// TwinCAT 3 PLC project Second_Floor_Totes_ARUP
// ProgramVersion: 3.1.4023.0
// libraries:
//   VisuElemMeter, * (System)
//   VisuElems, * (System)
//   VisuElemsSpecialControls, * (System)
//   VisuElemsWinControls, * (System)
//   VisuElemTextEditor, * (System)
//   VisuInputs, * (System)
//   VisuNativeControl, * (System)
//   Tc2_Standard, * (Beckhoff Automation GmbH)
//   Tc2_System, * (Beckhoff Automation GmbH)
//   Tc2_TcpIp, * (Beckhoff Automation GmbH)
//   Tc2_Utilities, * (Beckhoff Automation GmbH)
//   Tc3_Module, * (Beckhoff Automation GmbH)
// project tree:
//   DUTs/EAP/ E_EAP_PubType.TcDUT, ST_EAP_DEVICE.TcDUT (not stored), ST_EAP_Publisher.TcDUT, ST_EAP_Pub_Variable.TcDUT, ST_EAP_Subscriber.TcDUT (not stored), ST_EAP_Sub_Variable.TcDUT
//   DUTs/ E_EquipType.TcTLEO (not stored), E_StatusCode.TcDUT (not stored), ST_EquipmentStatus.TcDUT (not stored), ST_SafetyState.TcDUT (not stored)
//   DUTs/Messages/ E_EquipmentUpdate.TcTLEO (not stored), E_MessageIds.TcTLEO (not stored), E_TransportComplete.TcDUT (not stored), E_TransportResponse.TcTLEO (not stored), ST_Msg_ConveyorStat.TcDUT (not stored), ST_Msg_EquipStat.TcDUT (not stored)
//   / GlobalTextList.TcGTLO, PlcTask.TcTTO, Visualization Manager.TcVMO (not stored)
//   GVLs/ GVL_EquipArrays.TcGVL, GVL_IO.TcGVL, GVL_Logging.TcGVL, GVL_SorterItems.TcGVL, Onsite_Checklist.TcGVL
//   POUs/ BarCodeReaders.TcPOU, CommStatus.TcPOU, Conveyors.TcPOU, Log_Diverts.TcPOU, MAIN.TcPOU, MsgControl.TcPOU, Photoeyes.TcPOU, ProcessBuffers_6040.TcPOU, ProxSensors.TcPOU, P_PulseCountDist.TcPOU, ServerControl.TcPOU (not stored), Singulation_Control.TcPOU, Solenoids.TcPOU, Sorter.TcPOU, Sorter_P6040.TcPOU, System.TcPOU, SystemSafety.TcPOU
//   POUs/FunctionBlocks/BarCode/ CognexDataMan260.TcPOU (not stored)
//   POUs/FunctionBlocks/Binder/ BinderX_ReleaseControl.TcPOU (not stored), FB_BinderPusher.TcPOU (not stored), FB_Binder_SingulateHold.TcPOU (not stored)
//   POUs/FunctionBlocks/Binder/DUTs/ ST_Binder.TcDUT (not stored), ST_BinderState.TcDUT (not stored), ST_FromBinder.TcDUT (not stored), ST_ToBinder.TcDUT (not stored)
//   POUs/FunctionBlocks/Conveyance/DUTs/ E_ConvType.TcDUT (not stored)
//   POUs/FunctionBlocks/Conveyance/ FB_CnvyrCnfig_1.TcPOU, FB_SleepCntrl.TcPOU (not stored)
//   POUs/FunctionBlocks/Divert/DUTs/ ST_Divert.TcDUT, ST_DivertCfg.TcDUT
//   POUs/FunctionBlocks/Divert/Functions/ FB_ConfirmCheck.TcPOU (not stored), FB_DivertCommission.TcPOU, FB_DivertControl.TcPOU (not stored), FB_DivertDecision.TcPOU, FB_DivertFullMonitor.TcPOU (not stored), FB_DivertLog.TcPOU (not stored)
//   POUs/FunctionBlocks/Encoder/DUTs/ ST_Encoder.TcDUT (not stored)
//   POUs/FunctionBlocks/Encoder/ FB_ProcessEncoder.TcPOU (not stored)
//   POUs/FunctionBlocks/FB_Merge/ E_MergeState.TcDUT (not stored), FB_Merge2.TcPOU (not stored), MergeExample.TcPOU (not stored), ST_MergeSts.TcDUT (not stored)
//   POUs/FunctionBlocks/FB_Merge/Merge Inlet/ FB_MergeInlet.TcPOU (not stored), ST_MergeInlet.TcDUT (not stored), ST_MergeInletCfg.TcDUT (not stored), ST_MergeInletCtrl.TcDUT (not stored), ST_MergeInletSts.TcDUT (not stored)
//   POUs/FunctionBlocks/FB_MotionMerge/ FB_MotionMerge.TcPOU (not stored), MotionMergeExample.TcPOU (not stored), ST_MotionMergeConfig.TcDUT (not stored), ST_MotionMergeItem.TcDUT (not stored)
//   POUs/FunctionBlocks/Item/DUTs/ ST_Item.TcDUT (not stored), ST_ItemBuffer.TcDUT (not stored), ST_ItemBufferFdbk.TcDUT (not stored), ST_ItemLogBuffer.TcDUT (not stored), ST_ItemTemporary.TcDUT (not stored)
//   POUs/FunctionBlocks/Item/ FB_ItemBuffer.TcPOU (not stored), FB_ItemLogBuffer.TcPOU (not stored)
//   POUs/FunctionBlocks/LEDControl/ FB_LEDModeCtrl.TcPOU (not stored), ST_HMILEDMode.TcDUT (not stored), ST_LEDMode.TcDUT (not stored), ST_RGB.TcDUT (not stored)
//   POUs/FunctionBlocks/Logging/ FB_UpdateLog.TcPOU (not stored), ST_LogMsg.TcDUT (not stored)
//   POUs/FunctionBlocks/Metrics/ FB_Metrics.TcPOU (not stored)
//   POUs/FunctionBlocks/Server/Data types/ E_ConnectionSteps.TcDUT (not stored), E_ServerSteps.TcDUT (not stored)
//   POUs/FunctionBlocks/Server/ FB_Server.TcPOU (not stored), FB_ServerApplication.TcPOU (not stored), FB_ServerConnection.TcPOU (not stored)
//   POUs/FunctionBlocks/Server/Helper POUs/ FB_FrameFifo.TcPOU (not stored), FB_LogFifo.TcPOU (not stored)
//   POUs/FunctionBlocks/Singulation/ FB_Singulation.TcPOU (not stored)
//   POUs/FunctionBlocks/Solenoids/Functions/ FB_Solenoid_DA.TcPOU, FB_Solenoid_SA.TcPOU
//   POUs/FunctionBlocks/Sorter/DUTs/ ST_RoundRobin.TcDUT, ST_RoundRobinCfg.TcDUT (not stored), ST_RoundRobinDest.TcDUT (not stored), ST_Sorter.TcDUT, ST_SorterConfig.TcDUT
//   POUs/FunctionBlocks/Sorter/Functions/ FB_FindDestination.TcPOU, FB_SorterLog.TcPOU
//   POUs/FunctionBlocks/Sorter/ ProcessBuffers.TcPOU, SorterExample.TcPOU, SorterProgram.TcPOU (not stored)
//   POUs/FunctionBlocks/Sorter/VISUs/ ArrayInspection.TcVIS (not stored), DiverterTest.TcVIS (not stored), SorterArray.TcVIS
//   POUs/FunctionBlocks/StateControl/ E_OperStateCntrl.TcTLEO (not stored), E_StateCntrl.TcTLEO (not stored), E_StopCodes.TcTLEO (not stored), FB_ManageCodes.TcPOU (not stored), FB_StateCntrl.TcPOU (not stored), ST_StateCntrlPB.TcDUT (not stored), ST_StateCntrlSts.TcDUT (not stored)
//   POUs/FunctionBlocks/Utils/Events/ FB_EventMngr.TcPOU (not stored), FB_Intlks_Latch.TcPOU (not stored), FB_Intlks_NoLatch.TcPOU (not stored), ST_CfgEvents.TcDUT (not stored), ST_EventSts.TcDUT (not stored)
//   POUs/FunctionBlocks/Utils/ FB_AlrtStrtDelay.TcPOU (not stored), FB_EquipCntrl.TcPOU (not stored), FB_Flasher.TcPOU (not stored), FB_FlipFlop.TcPOU (not stored), FB_JamDetect.TcPOU (not stored), FB_PhotoEye.TcPOU (not stored), FB_SystemCntrl.TcPOU, F_CalculateDifference.TcPOU (not stored), F_CalculateIndex.TcPOU (not stored), F_DecIndex.TcPOU (not stored), F_IncIndex.TcPOU (not stored), F_PaddNumber.TcPOU (not stored), IncIndex.TcPOU (not stored), SystemCntrl_Example.TcPOU (not stored)
//   POUs/FunctionBlocks/Utils/Filters/ FB_DigDebnce.TcPOU, FB_DigDebnce_Off.TcPOU (not stored), FB_DigDebnce_On.TcPOU (not stored), F_Clip.TcPOU (not stored)
//   POUs/FunctionBlocks/VFD/DUTs/ DRIVE_STATE.TcTLEO (not stored)
//   POUs/FunctionBlocks/VFD/Functions/ DriveState.TcPOU (not stored), VFD.TcPOU
// real-time tasks:
//   TASK PlcTask: cycle T#10ms, priority 20, ADS port 350
//   TASK BCR_Sync: cycle T#1ms, priority 1, ADS port 301
// I/O:
//   DEVICE Device 1 (RT-Ethernet Protocol), AmsNetId 5.84.5.2.2.1
//   DEVICE Device 2 (TC3 EIP Scanner), AmsNetId 5.84.5.2.3.1
//     BCR_S6040_01 // <INFO> </INFO> <EDS> C:\TwinCAT\3.1\Config\Io\EtherNetIP\0678077313070100.eds </EDS>
//     BCR_S7004_01 // <INFO> </INFO> <EDS> C:\TwinCAT\3.1\Config\Io\EtherNetIP\0678077313070100.eds </EDS>
//   DEVICE Device 3 (EtherCAT), AmsNetId 5.84.5.2.4.1
//     Term 1 (EK1200) [EK1200-5000 EtherCAT Power supply (2A E-Bus)]
//       Term 2 (EL6070-0033) [EL6070-0033 1Ch. Licence key terminal, individual licences]
//       PLC-7021 (EL1008) [EL1008 8Ch. Dig. Input 24V, 3ms]
//       PLC-8051 (EL2008) [EL2008 8Ch. Dig. Output 24V, 0.5A]
//       PLC-8431 (EL1918) [EL1918, 8Ch. Safety Input 24V, TwinSAFE]
//         modules: Module 2 (FSLOGIC)
//       PLC-9071 (EL5152) [EL5152 2Ch. Inc. Encoder]
//       Term 7 (EK1122) [EK1122 2 port EtherCAT junction]
//         RIO-15181 (EP2339-0022) [EP2339-0022 16 Ch. Dig. Input/Output 24V, 0,5A, M12]
//         RIO-16171 (EP2339-0022) [EP2339-0022 16 Ch. Dig. Input/Output 24V, 0,5A, M12]
//         RIO-1181 (EP2339-0022) [EP2339-0022 16 Ch. Dig. Input/Output 24V, 0,5A, M12]
//         RIO-4172 (EP2339-0022) [EP2339-0022 16 Ch. Dig. Input/Output 24V, 0,5A, M12]
//         SRIO-5151 (EP1908) [EP1908, 8 Ch. Safety Input 24V, TwinSAFE ]
//           modules: Module 1 (FSOE)
//         RIO-6171 (EP2339-0022) [EP2339-0022 16 Ch. Dig. Input/Output 24V, 0,5A, M12]
//         RIO-7161 (EP2339-0022) [EP2339-0022 16 Ch. Dig. Input/Output 24V, 0,5A, M12]
//         RIO-8181 (EP2339-0022) [EP2339-0022 16 Ch. Dig. Input/Output 24V, 0,5A, M12]
//       Term 16 (EK1122) [EK1122 2 port EtherCAT junction]
//       Term 17 (EK1122) [EK1122 2 port EtherCAT junction]
//         SRIO-11141 (EP1908) [EP1908, 8 Ch. Safety Input 24V, TwinSAFE ]
//           modules: Module 1 (FSOE)
//         RIO-12171 (EP2339-0022) [EP2339-0022 16 Ch. Dig. Input/Output 24V, 0,5A, M12]
//         Term 18 (EK1100) [EK1100 EtherCAT Coupler (2A E-Bus)]
//           PLC-11021 (EL2008) [EL2008 8Ch. Dig. Output 24V, 0.5A]
//           PLC-11211 (EL2008) [EL2008 8Ch. Dig. Output 24V, 0.5A]
//           PLC-11431 (EL1008) [EL1008 8Ch. Dig. Input 24V, 3ms]
//           PLC-1008 (EL1008) [EL1008 8Ch. Dig. Input 24V, 3ms]
//           PLC-12061 (EL2008) [EL2008 8Ch. Dig. Output 24V, 0.5A]
//           PLC-12461 (EL1008) [EL1008 8Ch. Dig. Input 24V, 3ms]
//           PLC-13051 (EL1918) [EL1918, 8Ch. Safety Input 24V, TwinSAFE]
//             modules: Module 1 (FSOE), Module 2 (FSLOGIC)
//           PLC-13451 (EL2904) [EL2904, 4 Ch. Safety Output 24V, 0.5A, TwinSAFE]
//             modules: Module 1 (FSOES), Module 2 (DO)
//           Term 27 (EK1122) [EK1122 2 port EtherCAT junction]
//             P7040 (Inverter i550 Cabinet) [i550 Cabinet V05.04.xx]
//             P7005 (Inverter i550 Cabinet) [i550 Cabinet V05.04.xx]
//             P6010 (Inverter i550 Cabinet) [i550 Cabinet V05.04.xx]
//             P6045 (Inverter i550 Cabinet) [i550 Cabinet V05.04.xx]
//   DEVICE Communition with 205 (EtherCAT Automation Protocol), AmsNetId 5.84.5.2.5.1
//     Pub_To_205 (Publisher)
//     Sub_To_205 (Subscriber)
// variable links:
//   (this object) <-> Device 3 (EtherCAT)/Term 1 (EK1200)/PLC-8431 (EL1918)
//     Term 1 (EK1200)/Term 17 (EK1122)/SRIO-11141 (EP1908)/Module 1 (FSOE)/FSOE Inputs/FSOE <-> ConnectionOutputs/Message_33 RxPDO
//     Term 1 (EK1200)/Term 7 (EK1122)/SRIO-5151 (EP1908)/Module 1 (FSOE)/FSOE Inputs/FSOE <-> ConnectionOutputs/Message_32 RxPDO
//     Term 1 (EK1200)/Term 17 (EK1122)/SRIO-11141 (EP1908)/Module 1 (FSOE)/FSOE Outputs/FSOE <-> ConnectionInputs/Message_33 TxPDO
//     Term 1 (EK1200)/Term 7 (EK1122)/SRIO-5151 (EP1908)/Module 1 (FSOE)/FSOE Outputs/FSOE <-> ConnectionInputs/Message_32 TxPDO
//     Term 1 (EK1200)/Term 17 (EK1122)/Term 18 (EK1100)/PLC-13051 (EL1918)/Module 1 (FSOE)/FSoE Inputs/FSOE <-> ConnectionOutputs/Message_30 RxPDO
//     Term 1 (EK1200)/Term 17 (EK1122)/Term 18 (EK1100)/PLC-13051 (EL1918)/Module 1 (FSOE)/FSoE Outputs/FSOE <-> ConnectionInputs/Message_30 TxPDO
//     Term 1 (EK1200)/Term 17 (EK1122)/Term 18 (EK1100)/PLC-13451 (EL2904)/Module 1 (FSOES)/RxPDO/FSOE <-> ConnectionInputs/Message_31 TxPDO
//     Term 1 (EK1200)/Term 17 (EK1122)/Term 18 (EK1100)/PLC-13451 (EL2904)/Module 1 (FSOES)/TxPDO/FSOE <-> ConnectionOutputs/Message_31 RxPDO
//   (this object) <-> Device 3 (EtherCAT)/Term 1 (EK1200)/Term 17 (EK1122)/SRIO-11141 (EP1908)
//     Term 1 (EK1200)/PLC-8431 (EL1918)/ConnectionInputs/Message_33 TxPDO <-> Module 1 (FSOE)/FSOE Outputs/FSOE
//     Term 1 (EK1200)/PLC-8431 (EL1918)/ConnectionOutputs/Message_33 RxPDO <-> Module 1 (FSOE)/FSOE Inputs/FSOE
//   (this object) <-> Device 3 (EtherCAT)/Term 1 (EK1200)/Term 17 (EK1122)/Term 18 (EK1100)/PLC-13051 (EL1918)
//     Term 1 (EK1200)/PLC-8431 (EL1918)/ConnectionInputs/Message_30 TxPDO <-> Module 1 (FSOE)/FSoE Outputs/FSOE
//     Term 1 (EK1200)/PLC-8431 (EL1918)/ConnectionOutputs/Message_30 RxPDO <-> Module 1 (FSOE)/FSoE Inputs/FSOE
//   (this object) <-> Device 3 (EtherCAT)/Term 1 (EK1200)/Term 17 (EK1122)/Term 18 (EK1100)/PLC-13451 (EL2904)
//     Term 1 (EK1200)/PLC-8431 (EL1918)/ConnectionInputs/Message_31 TxPDO <-> Module 1 (FSOES)/RxPDO/FSOE
//     Term 1 (EK1200)/PLC-8431 (EL1918)/ConnectionOutputs/Message_31 RxPDO <-> Module 1 (FSOES)/TxPDO/FSOE
//   (this object) <-> Device 3 (EtherCAT)/Term 1 (EK1200)/Term 7 (EK1122)/SRIO-5151 (EP1908)
//     Term 1 (EK1200)/PLC-8431 (EL1918)/ConnectionInputs/Message_32 TxPDO <-> Module 1 (FSOE)/FSOE Outputs/FSOE
//     Term 1 (EK1200)/PLC-8431 (EL1918)/ConnectionOutputs/Message_32 RxPDO <-> Module 1 (FSOE)/FSOE Inputs/FSOE
//   Second_Floor_Totes_ARUP Instance <-> Communition with 205 (EtherCAT Automation Protocol)
//     PlcTask Inputs/MAIN.EAP_205.DevState <-> Inputs/DevState
//     PlcTask Outputs/MAIN.EAP_205.DevCtrl <-> Outputs/DevCtrl
//   Second_Floor_Totes_ARUP Instance <-> Communition with 205 (EtherCAT Automation Protocol)/Pub_To_205 (Publisher)
//     PlcTask Inputs/MAIN.EAP_205.Publisher.FrameState <-> Inputs/FrameState
//     PlcTask Inputs/MAIN.EAP_205.Publisher.Variables[0].VarState <-> To205_P6005_IsRunning/Inputs/VarState
//     PlcTask Inputs/MAIN.EAP_205.Publisher.Variables[1].VarState <-> To205_P7045_SendingProduct/Inputs/VarState
//     PlcTask Outputs/GVL_IO.To205_P6005_IsRunning <-> To205_P6005_IsRunning/Outputs/VarData
//     PlcTask Outputs/GVL_IO.To205_P7045_SendingProduct <-> To205_P7045_SendingProduct/Outputs/VarData
//     PlcTask Outputs/MAIN.EAP_205.Publisher.FrameCtrl <-> Outputs/FrameCtrl
//     PlcTask Outputs/MAIN.EAP_205.Publisher.IPAddr <-> Outputs/IpAddr
//     PlcTask Outputs/MAIN.EAP_205.Publisher.Variables[0].VarCtrl <-> To205_P6005_IsRunning/Outputs/VarCtrl
//     PlcTask Outputs/MAIN.EAP_205.Publisher.Variables[0].VarID <-> To205_P6005_IsRunning/Outputs/VarId
//     PlcTask Outputs/MAIN.EAP_205.Publisher.Variables[1].VarCtrl <-> To205_P7045_SendingProduct/Outputs/VarCtrl
//     PlcTask Outputs/MAIN.EAP_205.Publisher.Variables[1].VarID <-> To205_P7045_SendingProduct/Outputs/VarId
//   Second_Floor_Totes_ARUP Instance <-> Communition with 205 (EtherCAT Automation Protocol)/Sub_To_205 (Subscriber)
//     PlcTask Inputs/GVL_IO.From205_P2012_IsRunning <-> From205_P2012_IsRunning/Inputs/VarData
//     PlcTask Inputs/GVL_IO.From205_P3130_SendingProduct <-> From205_P3130_SendingProduct/Inputs/VarData
//     PlcTask Inputs/MAIN.EAP_205.Subscriber.FrameState <-> Inputs/FrameState
//     PlcTask Inputs/MAIN.EAP_205.Subscriber.Variables[0].CycleIndex <-> From205_P2012_IsRunning/Inputs/CycleIndex
//     PlcTask Inputs/MAIN.EAP_205.Subscriber.Variables[0].Quality <-> From205_P2012_IsRunning/Inputs/Quality
//     PlcTask Inputs/MAIN.EAP_205.Subscriber.Variables[0].VarState <-> From205_P2012_IsRunning/Inputs/VarState
//     PlcTask Inputs/MAIN.EAP_205.Subscriber.Variables[1].CycleIndex <-> From205_P3130_SendingProduct/Inputs/CycleIndex
//     PlcTask Inputs/MAIN.EAP_205.Subscriber.Variables[1].Quality <-> From205_P3130_SendingProduct/Inputs/Quality
//     PlcTask Inputs/MAIN.EAP_205.Subscriber.Variables[1].VarState <-> From205_P3130_SendingProduct/Inputs/VarState
//     PlcTask Outputs/MAIN.EAP_205.Subscriber.FrameCtrl <-> Outputs/FrameCtrl
//     PlcTask Outputs/MAIN.EAP_205.Subscriber.Variables[0].VarCtrl <-> From205_P2012_IsRunning/Outputs/VarCtrl
//     PlcTask Outputs/MAIN.EAP_205.Subscriber.Variables[0].VarId <-> From205_P2012_IsRunning/Outputs/VarId
//     PlcTask Outputs/MAIN.EAP_205.Subscriber.Variables[1].VarCtrl <-> From205_P3130_SendingProduct/Outputs/VarCtrl
//     PlcTask Outputs/MAIN.EAP_205.Subscriber.Variables[1].VarId <-> From205_P3130_SendingProduct/Outputs/VarId
//   Second_Floor_Totes_ARUP Instance <-> Device 1 (RT-Ethernet Protocol)
//     PlcTask Inputs/GVL_IO.EthernetAdapter_State <-> Inputs/DevState
//   Second_Floor_Totes_ARUP Instance <-> Device 2 (TC3 EIP Scanner)/BCR_S6040_01
//     PlcTask Inputs/BarCodeReaders.BCR_S6040_01.Acquiring <-> Connection 1 (Input/Output)/Inputs/Acquiring
//     PlcTask Inputs/BarCodeReaders.BCR_S6040_01.DecodeComplete <-> Connection 1 (Input/Output)/Inputs/Decode Complete
//     PlcTask Inputs/BarCodeReaders.BCR_S6040_01.Decoding <-> Connection 1 (Input/Output)/Inputs/Decoding
//     PlcTask Inputs/BarCodeReaders.BCR_S6040_01.DeviceState <-> Inputs/State
//     PlcTask Inputs/BarCodeReaders.BCR_S6040_01.ResultCode <-> Connection 1 (Input/Output)/Inputs/Result Code
//     PlcTask Inputs/BarCodeReaders.BCR_S6040_01.ResultData[0] <-> Connection 1 (Input/Output)/Inputs/Result Data
//     PlcTask Inputs/BarCodeReaders.BCR_S6040_01.ResultData[10] <-> Connection 1 (Input/Output)/Inputs/Result Data_10
//     PlcTask Inputs/BarCodeReaders.BCR_S6040_01.ResultData[11] <-> Connection 1 (Input/Output)/Inputs/Result Data_11
//     PlcTask Inputs/BarCodeReaders.BCR_S6040_01.ResultData[12] <-> Connection 1 (Input/Output)/Inputs/Result Data_12
//     PlcTask Inputs/BarCodeReaders.BCR_S6040_01.ResultData[13] <-> Connection 1 (Input/Output)/Inputs/Result Data_13
//     PlcTask Inputs/BarCodeReaders.BCR_S6040_01.ResultData[14] <-> Connection 1 (Input/Output)/Inputs/Result Data_14
//     PlcTask Inputs/BarCodeReaders.BCR_S6040_01.ResultData[15] <-> Connection 1 (Input/Output)/Inputs/Result Data_15
//     PlcTask Inputs/BarCodeReaders.BCR_S6040_01.ResultData[16] <-> Connection 1 (Input/Output)/Inputs/Result Data_16
//     PlcTask Inputs/BarCodeReaders.BCR_S6040_01.ResultData[1] <-> Connection 1 (Input/Output)/Inputs/Result Data_1
//     PlcTask Inputs/BarCodeReaders.BCR_S6040_01.ResultData[2] <-> Connection 1 (Input/Output)/Inputs/Result Data_2
//     PlcTask Inputs/BarCodeReaders.BCR_S6040_01.ResultData[3] <-> Connection 1 (Input/Output)/Inputs/Result Data_3
//     PlcTask Inputs/BarCodeReaders.BCR_S6040_01.ResultData[4] <-> Connection 1 (Input/Output)/Inputs/Result Data_4
//     PlcTask Inputs/BarCodeReaders.BCR_S6040_01.ResultData[5] <-> Connection 1 (Input/Output)/Inputs/Result Data_5
//     PlcTask Inputs/BarCodeReaders.BCR_S6040_01.ResultData[6] <-> Connection 1 (Input/Output)/Inputs/Result Data_6
//     PlcTask Inputs/BarCodeReaders.BCR_S6040_01.ResultData[7] <-> Connection 1 (Input/Output)/Inputs/Result Data_7
//     PlcTask Inputs/BarCodeReaders.BCR_S6040_01.ResultData[8] <-> Connection 1 (Input/Output)/Inputs/Result Data_8
//     PlcTask Inputs/BarCodeReaders.BCR_S6040_01.ResultData[9] <-> Connection 1 (Input/Output)/Inputs/Result Data_9
//     PlcTask Inputs/BarCodeReaders.BCR_S6040_01.ResultID <-> Connection 1 (Input/Output)/Inputs/Result ID
//     PlcTask Inputs/BarCodeReaders.BCR_S6040_01.ResultLength <-> Connection 1 (Input/Output)/Inputs/Result Length
//     PlcTask Inputs/BarCodeReaders.BCR_S6040_01.ResultsAvail <-> Connection 1 (Input/Output)/Inputs/Results Available
//     PlcTask Inputs/BarCodeReaders.BCR_S6040_01.TriggerAck <-> Connection 1 (Input/Output)/Inputs/Trigger Ack
//     PlcTask Inputs/BarCodeReaders.BCR_S6040_01.TriggerID <-> Connection 1 (Input/Output)/Inputs/Trigger ID
//     PlcTask Inputs/BarCodeReaders.BCR_S6040_01.TriggerReady <-> Connection 1 (Input/Output)/Inputs/Trigger Ready
//     PlcTask Outputs/BarCodeReaders.BCR_S6040_01.ResultsAck <-> Connection 1 (Input/Output)/Outputs/Results Ack
//     PlcTask Outputs/BarCodeReaders.BCR_S6040_01.Trigger <-> Connection 1 (Input/Output)/Outputs/Trigger
//     PlcTask Outputs/BarCodeReaders.BCR_S6040_01.TriggerEnable <-> Connection 1 (Input/Output)/Outputs/Trigger Enable
//   Second_Floor_Totes_ARUP Instance <-> Device 2 (TC3 EIP Scanner)/BCR_S7004_01
//     PlcTask Inputs/BarCodeReaders.BCR_S7004_01.Acquiring <-> Connection 2 (Input/Output)/Inputs/Acquiring
//     PlcTask Inputs/BarCodeReaders.BCR_S7004_01.DecodeComplete <-> Connection 2 (Input/Output)/Inputs/Decode Complete
//     PlcTask Inputs/BarCodeReaders.BCR_S7004_01.Decoding <-> Connection 2 (Input/Output)/Inputs/Decoding
//     PlcTask Inputs/BarCodeReaders.BCR_S7004_01.DeviceState <-> Inputs/State
//     PlcTask Inputs/BarCodeReaders.BCR_S7004_01.ResultCode <-> Connection 2 (Input/Output)/Inputs/Result Code
//     PlcTask Inputs/BarCodeReaders.BCR_S7004_01.ResultData[0] <-> Connection 2 (Input/Output)/Inputs/Result Data
//     PlcTask Inputs/BarCodeReaders.BCR_S7004_01.ResultData[10] <-> Connection 2 (Input/Output)/Inputs/Result Data_10
//     PlcTask Inputs/BarCodeReaders.BCR_S7004_01.ResultData[11] <-> Connection 2 (Input/Output)/Inputs/Result Data_11
//     PlcTask Inputs/BarCodeReaders.BCR_S7004_01.ResultData[12] <-> Connection 2 (Input/Output)/Inputs/Result Data_12
//     PlcTask Inputs/BarCodeReaders.BCR_S7004_01.ResultData[13] <-> Connection 2 (Input/Output)/Inputs/Result Data_13
//     PlcTask Inputs/BarCodeReaders.BCR_S7004_01.ResultData[14] <-> Connection 2 (Input/Output)/Inputs/Result Data_14
//     PlcTask Inputs/BarCodeReaders.BCR_S7004_01.ResultData[15] <-> Connection 2 (Input/Output)/Inputs/Result Data_15
//     PlcTask Inputs/BarCodeReaders.BCR_S7004_01.ResultData[16] <-> Connection 2 (Input/Output)/Inputs/Result Data_16
//     PlcTask Inputs/BarCodeReaders.BCR_S7004_01.ResultData[1] <-> Connection 2 (Input/Output)/Inputs/Result Data_1
//     PlcTask Inputs/BarCodeReaders.BCR_S7004_01.ResultData[2] <-> Connection 2 (Input/Output)/Inputs/Result Data_2
//     PlcTask Inputs/BarCodeReaders.BCR_S7004_01.ResultData[3] <-> Connection 2 (Input/Output)/Inputs/Result Data_3
//     PlcTask Inputs/BarCodeReaders.BCR_S7004_01.ResultData[4] <-> Connection 2 (Input/Output)/Inputs/Result Data_4
//     PlcTask Inputs/BarCodeReaders.BCR_S7004_01.ResultData[5] <-> Connection 2 (Input/Output)/Inputs/Result Data_5
//     PlcTask Inputs/BarCodeReaders.BCR_S7004_01.ResultData[6] <-> Connection 2 (Input/Output)/Inputs/Result Data_6
//     PlcTask Inputs/BarCodeReaders.BCR_S7004_01.ResultData[7] <-> Connection 2 (Input/Output)/Inputs/Result Data_7
//     PlcTask Inputs/BarCodeReaders.BCR_S7004_01.ResultData[8] <-> Connection 2 (Input/Output)/Inputs/Result Data_8
//     PlcTask Inputs/BarCodeReaders.BCR_S7004_01.ResultData[9] <-> Connection 2 (Input/Output)/Inputs/Result Data_9
//     PlcTask Inputs/BarCodeReaders.BCR_S7004_01.ResultID <-> Connection 2 (Input/Output)/Inputs/Result ID
//     PlcTask Inputs/BarCodeReaders.BCR_S7004_01.ResultLength <-> Connection 2 (Input/Output)/Inputs/Result Length
//     PlcTask Inputs/BarCodeReaders.BCR_S7004_01.ResultsAvail <-> Connection 2 (Input/Output)/Inputs/Results Available
//     PlcTask Inputs/BarCodeReaders.BCR_S7004_01.TriggerAck <-> Connection 2 (Input/Output)/Inputs/Trigger Ack
//     PlcTask Inputs/BarCodeReaders.BCR_S7004_01.TriggerID <-> Connection 2 (Input/Output)/Inputs/Trigger ID
//     PlcTask Inputs/BarCodeReaders.BCR_S7004_01.TriggerReady <-> Connection 2 (Input/Output)/Inputs/Trigger Ready
//     PlcTask Outputs/BarCodeReaders.BCR_S7004_01.ResultsAck <-> Connection 2 (Input/Output)/Outputs/Results Ack
//     PlcTask Outputs/BarCodeReaders.BCR_S7004_01.Trigger <-> Connection 2 (Input/Output)/Outputs/Trigger
//     PlcTask Outputs/BarCodeReaders.BCR_S7004_01.TriggerEnable <-> Connection 2 (Input/Output)/Outputs/Trigger Enable
//   Second_Floor_Totes_ARUP Instance <-> Device 3 (EtherCAT)/Term 1 (EK1200)/PLC-7021 (EL1008)
//     PlcTask Inputs/GVL_IO.PB_SysReset <-> Channel 3/Reset PB
//     PlcTask Inputs/GVL_IO.PB_SysStart <-> Channel 1/Start PB
//     PlcTask Inputs/GVL_IO.PB_SysStop <-> Channel 2/Stop PB
//   Second_Floor_Totes_ARUP Instance <-> Device 3 (EtherCAT)/Term 1 (EK1200)/PLC-8051 (EL2008)
//     PlcTask Outputs/GVL_IO.HornMainPanel <-> Channel 1/Horn
//     PlcTask Outputs/GVL_IO.LT_MainPanelStack_Green <-> Channel 4/LT-8111
//     PlcTask Outputs/GVL_IO.LT_MainPanelStack_Red <-> Channel 2/LT-8071
//     PlcTask Outputs/GVL_IO.LT_MainPanelStack_Yellow <-> Channel 3/LT-8091
//   Second_Floor_Totes_ARUP Instance <-> Device 3 (EtherCAT)/Term 1 (EK1200)/PLC-8431 (EL1918)
//     PlcTask Inputs/GVL_IO.PanelEstop_OK <-> StandardInputs/Standard Out Var 9
//     PlcTask Inputs/GVL_IO.Remote_PullCord6040_OK <-> StandardInputs/Standard Out Var 10
//     PlcTask Inputs/GVL_IO.Remote_PullCord7004_OK <-> StandardInputs/Standard Out Var 11
//     PlcTask Inputs/SystemSafety.Safety_SystemEstopsOK <-> StandardInputs/Standard Out Var 15
//     PlcTask Inputs/SystemSafety.SecondFloorShaft_Estop_OK <-> StandardInputs/Standard Out Var 36
//     PlcTask Inputs/SystemSafety.System_SafetyState.ComErr <-> StandardInputs/Standard Out Var 16
//     PlcTask Inputs/SystemSafety.System_SafetyState.FBErr <-> StandardInputs/Standard Out Var 17
//     PlcTask Inputs/SystemSafety.System_SafetyState.InRun <-> StandardInputs/Standard Out Var 38
//     PlcTask Inputs/SystemSafety.System_SafetyState.OtherErr <-> StandardInputs/Standard Out Var 18
//     PlcTask Inputs/SystemSafety.ThirdFloorShaft_Estop_OK <-> StandardInputs/Standard Out Var 37
//     PlcTask Outputs/SystemSafety.System_SafetyState.CommErrAck <-> StandardOutputs/Standard In Var 35
//     PlcTask Outputs/SystemSafety.System_SafetyState.ErrAck <-> StandardOutputs/Standard In Var 1
//     PlcTask Outputs/SystemSafety.System_SafetyState.Reset <-> StandardOutputs/Standard In Var 5
//     PlcTask Outputs/SystemSafety.System_SafetyState.Run <-> StandardOutputs/Standard In Var 2
//   Second_Floor_Totes_ARUP Instance <-> Device 3 (EtherCAT)/Term 1 (EK1200)/PLC-9071 (EL5152)
//     PlcTask Inputs/GVL_IO.ENC_9021_Period <-> ENC Period Channel 1/Period value
//     PlcTask Inputs/GVL_IO.ENC_9021_Raw <-> ENC Status compact Channel 1/Counter value
//   Second_Floor_Totes_ARUP Instance <-> Device 3 (EtherCAT)/Term 1 (EK1200)/Term 17 (EK1122)/RIO-12171 (EP2339-0022)
//     PlcTask Inputs/GVL_IO.DS_P7004 <-> Channel 9/P7004 Motor Disconnect
//     PlcTask Inputs/GVL_IO.DS_P7005 <-> Channel 8/P7005 Motor Discconnect
//     PlcTask Inputs/GVL_IO.DS_P7010 <-> Channel 11/P7010 Motor Discconnect
//     PlcTask Inputs/GVL_IO.PB_RemoteReset_12181 <-> Channel 4/PB-12181
//     PlcTask Inputs/GVL_IO.RIO12171_WcState <-> WcState/WcState
//     PlcTask Inputs/PhotoEyes.PE_12221.In_PE <-> Channel 5/PE-12221
//     PlcTask Inputs/PhotoEyes.PE_12261.In_PE <-> Channel 6/PE-12261
//     PlcTask Inputs/PhotoEyes.PE_12301.In_PE <-> Channel 7/PE-12301
//     PlcTask Inputs/PhotoEyes.PE_12231.In_PE <-> Channel 12/PE12231
//     PlcTask Outputs/GVL_IO.LT_12121_Red <-> Channel 17/LT-12121
//     PlcTask Outputs/GVL_IO.LT_12131_Yellow <-> Channel 18/LT-12131
//     PlcTask Outputs/GVL_IO.LT_12161_Green <-> Channel 19/LT-12161
//   Second_Floor_Totes_ARUP Instance <-> Device 3 (EtherCAT)/Term 1 (EK1200)/Term 17 (EK1122)/SRIO-11141 (EP1908)
//     PlcTask Inputs/GVL_IO.RIO11141_WcState <-> WcState/WcState
//   Second_Floor_Totes_ARUP Instance <-> Device 3 (EtherCAT)/Term 1 (EK1200)/Term 17 (EK1122)/Term 18 (EK1100)/PLC-1008 (EL1008)
//     PlcTask Inputs/GVL_IO.P6005_Faulted <-> Channel 1/P6005 Faulted
//     PlcTask Inputs/GVL_IO.P6015_Faulted <-> Channel 2/P6015 Faulted
//     PlcTask Inputs/GVL_IO.P6020_Faulted <-> Channel 3/P6020 Faulted
//     PlcTask Inputs/GVL_IO.P6025_Faulted <-> Channel 4/P6025 Faulted
//     PlcTask Inputs/GVL_IO.P6030_Faulted <-> Channel 5/P6030 Faulted
//     PlcTask Inputs/GVL_IO.P6035_Faulted <-> Channel 6/P6035 Faulted
//     PlcTask Inputs/GVL_IO.P6040_Faulted <-> Channel 7/P6040 Faulted
//   Second_Floor_Totes_ARUP Instance <-> Device 3 (EtherCAT)/Term 1 (EK1200)/Term 17 (EK1122)/Term 18 (EK1100)/PLC-11021 (EL2008)
//     PlcTask Outputs/GVL_IO.P7004_RUN <-> Channel 1/P7004 RUN
//     PlcTask Outputs/GVL_IO.P7010_RUN <-> Channel 2/P7010 RUN
//     PlcTask Outputs/GVL_IO.P7015_RUN <-> Channel 3/P7015 RUN
//     PlcTask Outputs/GVL_IO.P7020_RUN <-> Channel 4/P7020 RUN
//     PlcTask Outputs/GVL_IO.P7025_RUN <-> Channel 5/P7025 RUN
//     PlcTask Outputs/GVL_IO.P7030_RUN <-> Channel 6/P7030 RUN
//     PlcTask Outputs/GVL_IO.P7035_RUN <-> Channel 7/P7035 RUN
//     PlcTask Outputs/GVL_IO.P7045_RUN <-> Channel 8/P7045 RUN
//   Second_Floor_Totes_ARUP Instance <-> Device 3 (EtherCAT)/Term 1 (EK1200)/Term 17 (EK1122)/Term 18 (EK1100)/PLC-11211 (EL2008)
//     PlcTask Outputs/GVL_IO.P6005_RUN <-> Channel 1/P6005 RUN
//     PlcTask Outputs/GVL_IO.P6015_RUN <-> Channel 2/P6015 RUN
//     PlcTask Outputs/GVL_IO.P6020_RUN <-> Channel 3/P6020 RUN
//     PlcTask Outputs/GVL_IO.P6025_RUN <-> Channel 4/P6025 RUN
//     PlcTask Outputs/GVL_IO.P6030_RUN <-> Channel 5/P6030 RUN
//     PlcTask Outputs/GVL_IO.P6035_RUN <-> Channel 6/P6035 RUN
//     PlcTask Outputs/GVL_IO.P6040_RUN <-> Channel 7/P6040 RUN
//   Second_Floor_Totes_ARUP Instance <-> Device 3 (EtherCAT)/Term 1 (EK1200)/Term 17 (EK1122)/Term 18 (EK1100)/PLC-11431 (EL1008)
//     PlcTask Inputs/GVL_IO.P7004_Faulted <-> Channel 1/P7004 Faulted
//     PlcTask Inputs/GVL_IO.P7010_Faulted <-> Channel 2/P7010 Faulted
//     PlcTask Inputs/GVL_IO.P7015_Faulted <-> Channel 3/P7015 Faulted
//     PlcTask Inputs/GVL_IO.P7020_Faulted <-> Channel 4/P7020 Faulted
//     PlcTask Inputs/GVL_IO.P7025_Faulted <-> Channel 5/P7025 Faulted
//     PlcTask Inputs/GVL_IO.P7030_Faulted <-> Channel 6/P7030 Faulted
//     PlcTask Inputs/GVL_IO.P7035_Faulted <-> Channel 7/P7035 Faulted
//     PlcTask Inputs/GVL_IO.P7045_Faulted <-> Channel 8/P7045 Faulted
//   Second_Floor_Totes_ARUP Instance <-> Device 3 (EtherCAT)/Term 1 (EK1200)/Term 17 (EK1122)/Term 18 (EK1100)/Term 27 (EK1122)/P6010 (Inverter i550 Cabinet)
//     PlcTask Inputs/Conveyors.P6010_VFD.ActualVelocity <-> TPDO (A) Velocity/Actual speed
//     PlcTask Inputs/Conveyors.P6010_VFD.StatusWord <-> TPDO (A) Velocity/CiA status word
//     PlcTask Outputs/Conveyors.P6010_VFD.ControlWord <-> RPDO (A) Velocity/CiA control word
//     PlcTask Outputs/Conveyors.P6010_VFD.TargetVelocity <-> RPDO (A) Velocity/Set speed
//   Second_Floor_Totes_ARUP Instance <-> Device 3 (EtherCAT)/Term 1 (EK1200)/Term 17 (EK1122)/Term 18 (EK1100)/Term 27 (EK1122)/P6045 (Inverter i550 Cabinet)
//     PlcTask Inputs/Conveyors.P6045_VFD.ActualVelocity <-> TPDO (A) Velocity/Actual speed
//     PlcTask Inputs/Conveyors.P6045_VFD.StatusWord <-> TPDO (A) Velocity/CiA status word
//     PlcTask Outputs/Conveyors.P6045_VFD.ControlWord <-> RPDO (A) Velocity/CiA control word
//     PlcTask Outputs/Conveyors.P6045_VFD.TargetVelocity <-> RPDO (A) Velocity/Set speed
//   Second_Floor_Totes_ARUP Instance <-> Device 3 (EtherCAT)/Term 1 (EK1200)/Term 17 (EK1122)/Term 18 (EK1100)/Term 27 (EK1122)/P7005 (Inverter i550 Cabinet)
//     PlcTask Inputs/Conveyors.P7005_VFD.ActualVelocity <-> TPDO (A) Velocity/Actual speed
//     PlcTask Inputs/Conveyors.P7005_VFD.StatusWord <-> TPDO (A) Velocity/CiA status word
//     PlcTask Outputs/Conveyors.P7005_VFD.ControlWord <-> RPDO (A) Velocity/CiA control word
//     PlcTask Outputs/Conveyors.P7005_VFD.TargetVelocity <-> RPDO (A) Velocity/Set speed
//   Second_Floor_Totes_ARUP Instance <-> Device 3 (EtherCAT)/Term 1 (EK1200)/Term 17 (EK1122)/Term 18 (EK1100)/Term 27 (EK1122)/P7040 (Inverter i550 Cabinet)
//     PlcTask Inputs/Conveyors.P7040_VFD.ActualVelocity <-> TPDO (A) Velocity/Actual speed
//     PlcTask Inputs/Conveyors.P7040_VFD.StatusWord <-> TPDO (A) Velocity/CiA status word
//     PlcTask Outputs/Conveyors.P7040_VFD.ControlWord <-> RPDO (A) Velocity/CiA control word
//     PlcTask Outputs/Conveyors.P7040_VFD.TargetVelocity <-> RPDO (A) Velocity/Set speed
//   Second_Floor_Totes_ARUP Instance <-> Device 3 (EtherCAT)/Term 1 (EK1200)/Term 7 (EK1122)/RIO-1181 (EP2339-0022)
//     PlcTask Inputs/GVL_IO.DS_P6005 <-> Channel 14/P6005 Motor Disconnect
//     PlcTask Inputs/GVL_IO.DS_P6015 <-> Channel 10/P6015 Motor Disconnect
//     PlcTask Inputs/GVL_IO.DS_P6010 <-> Channel 12/P6010 Motor Disconnect
//     PlcTask Inputs/GVL_IO.DS_P6020 <-> Channel 4/P6020 Dissconnect
//     PlcTask Inputs/GVL_IO.RIO1181_WcState <-> WcState/WcState
//     PlcTask Inputs/PhotoEyes.PE_1081.In_PE <-> Channel 9/PE-1081
//     PlcTask Inputs/PhotoEyes.PE_1161.In_PE <-> Channel 3/PE-1161
//     PlcTask Inputs/PhotoEyes.PE_1162.In_PE <-> Channel 11/PE-1162
//     PlcTask Inputs/PhotoEyes.PE_1231.In_PE <-> Channel 5/PE-1231
//     PlcTask Inputs/PhotoEyes.PE_1232.In_PE <-> Channel 13/PE-1232
//     PlcTask Inputs/ProxSensors.In_PX_1281_Extended <-> Channel 6/PX-1281
//   Second_Floor_Totes_ARUP Instance <-> Device 3 (EtherCAT)/Term 1 (EK1200)/Term 7 (EK1122)/RIO-15181 (EP2339-0022)
//     PlcTask Inputs/GVL_IO.DS_P7015 <-> Channel 2/P7015 Motor Disconnect
//     PlcTask Inputs/GVL_IO.DS_P7020 <-> Channel 4/P7020 Motor Disconnect
//     PlcTask Inputs/GVL_IO.DS_P7025 <-> Channel 6/P7025 Motor Disconnect
//     PlcTask Inputs/GVL_IO.RIO15181_WcState <-> WcState/WcState
//     PlcTask Inputs/PhotoEyes.PE_15121.In_PE <-> Channel 1/PE-15121
//     PlcTask Inputs/PhotoEyes.PE_15181.In_PE <-> Channel 3/PE-15181
//     PlcTask Inputs/PhotoEyes.PE_15261.In_PE <-> Channel 5/PE-15261
//   Second_Floor_Totes_ARUP Instance <-> Device 3 (EtherCAT)/Term 1 (EK1200)/Term 7 (EK1122)/RIO-16171 (EP2339-0022)
//     PlcTask Inputs/GVL_IO.DS_P7030 <-> Channel 2/P7030 Motor Disconnect
//     PlcTask Inputs/GVL_IO.DS_P7035 <-> Channel 8/P7035 Motor Discconnect
//     PlcTask Inputs/GVL_IO.DS_P7040 <-> Channel 10/P7040 Motor Discconnect
//     PlcTask Inputs/GVL_IO.DS_P7045 <-> Channel 12/P7045 Motor discconnect
//     PlcTask Inputs/GVL_IO.RIO16171_WcState <-> WcState/WcState
//     PlcTask Inputs/PhotoEyes.PE_16111.In_PE <-> Channel 1/PE-16111
//     PlcTask Inputs/PhotoEyes.PE_16131.In_PE <-> Channel 9/PE-16131
//     PlcTask Inputs/PhotoEyes.PE_16181.In_PE <-> Channel 3/PE-16181
//     PlcTask Inputs/PhotoEyes.PE_16201.In_PE <-> Channel 11/PE-16201
//     PlcTask Inputs/PhotoEyes.PE_16301.In_PE <-> Channel 7/PE-16301
//     PlcTask Inputs/ProxSensors.In_PX_16231_Extended <-> Channel 5/PX-16231
//   Second_Floor_Totes_ARUP Instance <-> Device 3 (EtherCAT)/Term 1 (EK1200)/Term 7 (EK1122)/RIO-4172 (EP2339-0022)
//     PlcTask Inputs/GVL_IO.DS_P6025 <-> Channel 10/P6025 Motor disconnect
//     PlcTask Inputs/GVL_IO.DS_P6030 <-> Channel 8/P6030 Motor Discconnect
//     PlcTask Inputs/GVL_IO.DS_P6035 <-> Channel 6/P6035 Motor Disconnect
//     PlcTask Inputs/GVL_IO.DS_P6045 <-> Channel 2/P6045 Motor Discconnect
//     PlcTask Inputs/GVL_IO.RIO4172_WcState <-> WcState/WcState
//     PlcTask Inputs/PhotoEyes.PE_4071.In_PE <-> Channel 1/PE-4071
//     PlcTask Inputs/PhotoEyes.PE_4121.In_PE <-> Channel 9/PE-4121
//     PlcTask Inputs/PhotoEyes.PE_4201.In_PE <-> Channel 5/PE-4201
//     PlcTask Inputs/PhotoEyes.PE_4271.In_PE <-> Channel 7/PE-4271
//   Second_Floor_Totes_ARUP Instance <-> Device 3 (EtherCAT)/Term 1 (EK1200)/Term 7 (EK1122)/RIO-6171 (EP2339-0022)
//     PlcTask Inputs/GVL_IO.RIO6171_WcState <-> WcState/WcState
//     PlcTask Inputs/PhotoEyes.PE_6181.In_PE <-> Channel 11/PE-6181
//     PlcTask Inputs/PhotoEyes.PE_6201.In_PE <-> Channel 12/PE-6201
//     PlcTask Inputs/PhotoEyes.PE_6241.In_PE <-> Channel 13/PE-6241
//     PlcTask Inputs/PhotoEyes.PE_6261.In_PE <-> Channel 14/PE-6261
//     PlcTask Inputs/PhotoEyes.PE_6302.In_PE <-> Channel 15/PE-6302
//     PlcTask Inputs/ProxSensors.In_PX_6121_Retracted <-> Channel 1/PX-6121
//     PlcTask Inputs/ProxSensors.In_PX_6122_Retracted <-> Channel 9/PX-6122
//     PlcTask Inputs/ProxSensors.In_PX_6241_Retracted <-> Channel 5/PX-6241
//     PlcTask Inputs/ProxSensors.In_PX_6151_Extended <-> Channel 2/PX-6151
//     PlcTask Inputs/ProxSensors.In_PX_6152_Extended <-> Channel 10/PX-6152
//     PlcTask Inputs/ProxSensors.In_PX_6261_Extended <-> Channel 6/PX-6261
//     PlcTask Outputs/GVL_IO.SV_6181_EXT <-> Channel 19/SV-6181
//     PlcTask Outputs/GVL_IO.SV_6211_EXT <-> Channel 20/SV-6211
//     PlcTask Outputs/GVL_IO.SV_6321_EXT <-> Channel 24/SV-6321
//     PlcTask Outputs/GVL_IO.SV_6301_RET <-> Channel 23/SV-6301
//   Second_Floor_Totes_ARUP Instance <-> Device 3 (EtherCAT)/Term 1 (EK1200)/Term 7 (EK1122)/RIO-7161 (EP2339-0022)
//     PlcTask Inputs/GVL_IO.PB_RemoteReset_7281 <-> Channel 16/PB-7281
//     PlcTask Inputs/GVL_IO.RIO7161_WcState <-> WcState/WcState
//     PlcTask Inputs/PhotoEyes.PE_7151.In_PE <-> Channel 10/PE-7151
//     PlcTask Inputs/PhotoEyes.PE_7191.In_PE <-> Channel 11/PE-7191
//     PlcTask Inputs/PhotoEyes.PE_7211.In_PE <-> Channel 4/PE-7211
//     PlcTask Inputs/PhotoEyes.PE_7241.In_PE <-> Channel 5/PE-7241
//     PlcTask Inputs/PhotoEyes.PE_7171.In_PE <-> Channel 12/PE7171
//     PlcTask Inputs/ProxSensors.In_PX_7122_Retracted <-> Channel 1/PX-7122
//     PlcTask Inputs/ProxSensors.In_PX_7271_Retracted <-> Channel 7/PX-7271
//     PlcTask Inputs/ProxSensors.In_PX_7151_Extended <-> Channel 2/PX-7151
//     PlcTask Inputs/ProxSensors.In_PX_7301_Extended <-> Channel 8/PX-7301
//     PlcTask Outputs/GVL_IO.LT_7221_Red <-> Channel 29/LT-7221
//     PlcTask Outputs/GVL_IO.LT_7241_Yellow <-> Channel 30/LT-7241
//     PlcTask Outputs/GVL_IO.LT_7271_Green <-> Channel 31/LT-7271
//     PlcTask Outputs/GVL_IO.SV_7121_EXT <-> Channel 25/SV-7121
//     PlcTask Outputs/GVL_IO.SV_7181_EXT <-> Channel 19/SV-7181
//   Second_Floor_Totes_ARUP Instance <-> Device 3 (EtherCAT)/Term 1 (EK1200)/Term 7 (EK1122)/RIO-8181 (EP2339-0022)
//     PlcTask Inputs/GVL_IO.DS_P6040 <-> Channel 6/P6040 Motor Disconnect
//     PlcTask Inputs/GVL_IO.RIO8181_WcState <-> WcState/WcState
//     PlcTask Inputs/GVL_IO.SystemAirPressure <-> Channel 15/Air Switch
//     PlcTask Inputs/PhotoEyes.PE_8141.In_PE <-> Channel 10/PE-8141
//     PlcTask Inputs/PhotoEyes.PE_8171.In_PE <-> Channel 11/PE-8171
//     PlcTask Inputs/PhotoEyes.PE_8181.In_PE <-> Channel 4/PE-8181
//     PlcTask Inputs/PhotoEyes.PE_8211.In_PE <-> Channel 13/PE-8211
//     PlcTask Inputs/PhotoEyes.PE_8221.In_PE <-> Channel 5/PE-8221
//     PlcTask Inputs/ProxSensors.In_PX_8091_Retracted <-> Channel 1/PX-8091
//     PlcTask Inputs/ProxSensors.In_PX_8321_Retracted <-> Channel 8/PX-8321
//     PlcTask Inputs/ProxSensors.In_PX_8121_Extended <-> Channel 2/PX-8121
//     PlcTask Inputs/ProxSensors.In_PX_8291_Extended <-> Channel 7/PX-8291
//     PlcTask Outputs/GVL_IO.SV_8111_EXT <-> Channel 25/SV-8111
//     PlcTask Outputs/GVL_IO.SV_8161_EXT <-> Channel 19/SV-8161
//   Second_Floor_Totes_ARUP Instance <-> Device 3 (EtherCAT)/Term 1 (EK1200)/Term 7 (EK1122)/SRIO-5151 (EP1908)
//     PlcTask Inputs/GVL_IO.RIO5151_WcState <-> WcState/WcState

CONFIGURATION Second_Floor_Totes_ARUP
    RESOURCE PLC ON TwinCAT3
        TASK PlcTask(INTERVAL := T#10ms, PRIORITY := 20);
        PROGRAM MAIN WITH PlcTask : MAIN;
    END_RESOURCE
END_CONFIGURATION

// ---- DUTs/EAP/E_EAP_PubType.TcDUT
{attribute 'qualified_only'}
{attribute 'strict'}
TYPE E_EAP_PubType :
(
	e_AmsNetID 	:= 0,
	e_IPAddr	:= 1,
	e_MAC_ID	:= 2
);
END_TYPE

// ---- DUTs/EAP/ST_EAP_Publisher.TcDUT
TYPE ST_EAP_Publisher :
STRUCT
	Name				: 	STRING;		// Name of the EAP Publisher
	FrameState	AT %I*	: 	UINT;		// EAP FrameState, FrameState.0 = Not Transmitting, .1 = Frame too large, .2 = Subscriber Miissing
	FrameCtrl	AT %Q*	: 	UINT;		// EAP FrameCtrl, FrameCtrl.0 = Disable Sending, .1 = Remove destination MAC from ARP
	PubType				:	E_EAP_PubType := 0;	// EAP Publisher Type, AMS NetID (0), IP Address (1), MAC ID (2)
	NetID		AT %Q*	: 	AMSNETID;	// EAP Changeable NetID
	IPAddr		AT %Q*	: 	UDINT;		// EAP Changeable IP, stored as a single UDINT
	HMI_IPAddr			: 	USINTARR4;	// Used to enter IP Address on the HMI, MEMCPY function copies array to IPAddr 
	HMI_IPAddrDisp		: 	USINTARR4;	// Used to Display IP Address on the HMI, MEMCPY function copies IPAddr to Array 
	MACID		AT %Q*	: 	USINTARR6;	// EAP Changeable MAC ID, stored as an array of 6 USINT
	Variables			:	ARRAY[0..9] OF ST_EAP_Pub_Variable;		// Array of Published variables
END_STRUCT
END_TYPE

// ---- DUTs/EAP/ST_EAP_Pub_Variable.TcDUT
TYPE ST_EAP_Pub_Variable :
STRUCT
	Name				: 	STRING;		// Name of the Variable
	VarState	AT %I*	:	UINT;		// VarState.0 = Not Sent, 1 = Transmission Suspended, 0 = Transmission OK
	VarID 		AT %Q*	:	UINT;		// Changeable ID of the variable
	VarCtrl		AT %Q*	:	UINT;		// VarCtrl.0 = Disable publishing
END_STRUCT
END_TYPE

// ---- DUTs/EAP/ST_EAP_Sub_Variable.TcDUT
TYPE ST_EAP_Sub_Variable :
STRUCT
	Name				: 	STRING;		// Name of the Variable
	VarState	AT %I*	:	UINT;		// VarState.0 = Invalid Hash/Version, .1 = Invalid Variable Length
	Quality		AT %I*	:	UINT;		// <>0, Duration the variable is not refreshed (in 100µs)
	CycleIndex	AT %I*	:	UINT;		// Incremented each publisher cycle
	VarId		AT %Q*	:	UINT;		// Changable Variable ID
	VarCtrl		AT %Q*	:	UINT;		// VarCtrl.1 = Ignore Hash/Version
END_STRUCT
END_TYPE

// ---- POUs/FunctionBlocks/Divert/DUTs/ST_Divert.TcDUT
TYPE ST_Divert :
{attribute 'OPC.UA.DA' := '1'}
STRUCT
	{attribute 'OPC.UA.DA' := '0'}
	Config			: ST_DivertCfg;		// Configuration Variables

	Full 			: BOOL;				//Diverter full photo eye is blocked
	Jammed 			: BOOL;				//Jammed photo eye is blocked
	Faulted 		: BOOL;				//Returned faulted status
	Status 			: E_StatusCode := E_StatusCode.Divert_Idle; 	//Status Code, initialized to Idle

	ConfirmPE	   	: BOOL;				//Physical input address of photo eye
	FullPE		   	: BOOL;				//Physical input address of photo eye
	JamPE		   	: BOOL;				//Physical input address of photo eye 
	Output1	 		: BOOL;				//Physical output address of diverter
	Output2	  		: BOOL;				//Physical output address of diverter
	
	{attribute 'OPC.UA.DA' := '0'}
	Output1Flag		: DINT;				//Indicates what the encoder count is when output is energized
	
	FullTime		: TIME;				//Time that full PE has to be high before the lane is considered full     
	{attribute 'OPC.UA.DA' := '0'}
	FullTimer		: TON; 				//Timer that is used for checking how long the full PE is on
	
	{attribute 'OPC.UA.DA' := '0'}
	Item			: ST_Item;			// Currently Diverting Item
END_STRUCT
END_TYPE

// ---- POUs/FunctionBlocks/Divert/DUTs/ST_DivertCfg.TcDUT
TYPE ST_DivertCfg :
{attribute 'OPC.UA.DA' := '1'}
STRUCT
	ID 				: STRING;			// User assigned Divert indetifier		
	EquipID 		: STRING[5];		// Identifier used for host communication		
	Number			: INT;				// Divert number, can be distinct from the Index in the Divert Array
	Distance		: INT;				// Distance, in encoder counts, from induct photo eye
	ConfirmDist		: INT;				// Distance from the Divert point to the Confirm PE
	Direction		: BOOL;				// 0 = Divert to one side, 1 = Divert to the other side 
	FullTime		: REAL;				// Time, in seconds, that full PE has to be high before the lane is considered full
	IsDischarge		: BOOL;				// TRUE, process and test for items destined for non-discharge diverts that missed
END_STRUCT
END_TYPE

// ---- POUs/FunctionBlocks/Sorter/DUTs/ST_RoundRobin.TcDUT
TYPE ST_RoundRobin :
{attribute 'OPC.UA.DA' := '1'}
STRUCT
	Destination		:	DINT;
	Enabled			:	UINT;
	Available		:	UINT;
	Sent			:	UINT;
	aDestinations	:	ARRAY[0..32] OF DINT;
END_STRUCT
END_TYPE

// ---- POUs/FunctionBlocks/Sorter/DUTs/ST_Sorter.TcDUT
TYPE ST_Sorter :
{attribute 'OPC.UA.DA' := '1'}
STRUCT
	{attribute 'OPC.UA.DA' := '0'}
	Config				: ST_SorterConfig;
	InductPE			: BOOL;
	EncoderCounts		: UDINT;
	LastUniqueID		: UINT;
	DischargePE			: BOOL;
END_STRUCT
END_TYPE

// ---- POUs/FunctionBlocks/Sorter/DUTs/ST_SorterConfig.TcDUT
TYPE ST_SorterConfig :
{attribute 'OPC.UA.DA' := '1'}
STRUCT
	Name				: STRING[5];
	EquipID				: STRING[5];
	Length				: UINT;
	InductWindow		: UINT;
	MinimumLength		: UINT;
	TailEndLength 		: UINT;
	Output2Offset		: UINT;
	DefaultDestination 	: DINT;
	DefaultDestIdx		: DINT;
	RecircDestination 	: DINT;
	RecircDestIdx 		: DINT;
	RecircUsed			: BOOL;
	RetainOnRestart		: BOOL;
	DivertCount			: DINT;
	RoundRobin			: ST_RoundRobin;
END_STRUCT
END_TYPE

// ---- GVLs/GVL_EquipArrays.TcGVL
{attribute 'qualified_only'}
VAR_GLOBAL
	nEquipIndex : DINT := 0;	// Index used to Assign the Equipment Index for System Status Reporting
	nEquip_Count AT %Q* : DINT; //Count of Equipment to Process in System PLC
	aEquipStatusArray_Out AT %Q* : ARRAY[1..cEQUIP_COUNT_MAX] OF ST_StateCntrlSts; //Array of Equipment Status Outbound
	aEquipStatusArray_In AT %I* : ARRAY[1..cEQUIP_COUNT_MAX] OF ST_StateCntrlSts; //Array of Equipment Status Inbound
	
	// OCR Equipment
	nOCREquip_Count AT %I* : DINT; //Count of Equipment to Process in System PLC
	aOCREquipStatusArray_Out AT %Q* : ARRAY[1..cEQUIP_COUNT_MAX] OF ST_StateCntrlSts; //Array of Equipment Status Outbound
	aOCREquipStatusArray_In AT %I* : ARRAY[1..cEQUIP_COUNT_MAX] OF ST_StateCntrlSts; //Array of Equipment Status Inbound
	// InspctCnvyr Equipment
	nInspctCnvyrEquip_Count AT %I* : DINT; //Count of Equipment to Process in System PLC
	aInspctCnvyrEquipStatusArray_Out AT %Q* : ARRAY[1..cEQUIP_COUNT_MAX] OF ST_StateCntrlSts; //Array of Equipment Status Outbound
	aInspctCnvyrEquipStatusArray_In AT %I* : ARRAY[1..cEQUIP_COUNT_MAX] OF ST_StateCntrlSts; //Array of Equipment Status Inbound
	// Sorter Equipment
	nSorterEquip_Count AT %I* : DINT; //Count of Equipment to Process in System PLC
	aSorterEquipStatusArray_Out AT %Q* : ARRAY[1..cEQUIP_COUNT_MAX] OF ST_StateCntrlSts; //Array of Equipment Status Outbound
	aSorterEquipStatusArray_In AT %I* : ARRAY[1..cEQUIP_COUNT_MAX] OF ST_StateCntrlSts; //Array of Equipment Status Inbound
	// System Equipment
	nSystemEquip_Count : DINT; //Count of Equipment to Process in System PLC
	aSystemEquipStatusArray : ARRAY[1..cEQUIP_COUNT_MAX] OF ST_StateCntrlSts; //Array of Equipment Status Current
	aSystemEquipStatusArray_Last : ARRAY[1..cEQUIP_COUNT_MAX] OF ST_StateCntrlSts; //Array of Equipment Status Last State
END_VAR

VAR_GLOBAL CONSTANT
	cEQUIP_COUNT_MAX : DINT := 25;	//Adjust when adding equipment to monitor
END_VAR

// ---- GVLs/GVL_IO.TcGVL
{attribute 'qualified_only'}
VAR_GLOBAL
	INIT						: BOOL := TRUE;		// Initialization Bit
	
	PB_SysStart AT %I* 		:BOOL;		//System Start Button
	PB_SysStop	AT %I*		:BOOL;		//System Stop Button
	PB_SysReset	AT %I* 		:BOOL; 		//System Reset Button
	PB_RemoteReset_7281 AT %I*		: BOOL;	//P6040 Reset Button
 	PB_RemoteReset_12181 AT %I* 	: BOOL;	//P7004 Height check reset Reset Button
	
	SystemAirPressure AT %I*	:BOOL;
	Regulator_AirPressure AT %I*	:BOOL;

	
	HornMainPanel				AT %Q* 	:BOOL;	//Panel Tower Horn
	{attribute 'OPC.UA.DA' := '1'}
	LT_MainPanelStack_Red		AT %Q*	:BOOL;	//Panel	Tower Red Light
	{attribute 'OPC.UA.DA' := '1'}
	LT_MainPanelStack_Yellow	AT %Q*	:BOOL;	//Panel	Tower Yellow Light
	{attribute 'OPC.UA.DA' := '1'}
	LT_MainPanelStack_Green		AT %Q*	:BOOL;	//Panel	Tower Green Light

	{attribute 'OPC.UA.DA' := '1'}
	LT_7221_Red	    AT %Q*	:BOOL;	//Panel	Tower Red Light
	{attribute 'OPC.UA.DA' := '1'}
	LT_7241_Yellow	AT %Q*	:BOOL;	//Panel	Tower Yellow Light
	{attribute 'OPC.UA.DA' := '1'}
	LT_7271_Green	AT %Q*	:BOOL;	//Panel	Tower Green Light
	
	{attribute 'OPC.UA.DA' := '1'}
	LT_12121_Red	AT %Q*	:BOOL;	//Panel	Tower Red Light
	{attribute 'OPC.UA.DA' := '1'}
	LT_12131_Yellow	AT %Q*	:BOOL;	//Panel	Tower Yellow Light
	{attribute 'OPC.UA.DA' := '1'}
	LT_12161_Green	AT %Q*	:BOOL;	//Panel	Tower Green Light
	
	{attribute 'OPC.UA.DA' := '1'}
	PanelEstop_OK AT %I* : BOOL;
	{attribute 'OPC.UA.DA' := '1'}
	Remote_PullCord6040_OK AT %I*: BOOL;
	{attribute 'OPC.UA.DA' := '1'}
	Remote_PullCord7004_OK AT %I*: BOOL;
	
//---------------------------------Motor Outputs-------------------------------------------------	

P6005_RUN            AT %Q*   :BOOL;    //P6005 Run Command
P6015_RUN            AT %Q*   :BOOL;    //P6015 Run Command
P6020_RUN            AT %Q*   :BOOL;    //P6020 Run Command
P6025_RUN            AT %Q*   :BOOL;    //P6025 Run Command
P6030_RUN            AT %Q*   :BOOL;    //P6030 Run Command
P6035_RUN            AT %Q*   :BOOL;    //P6035 Run Command
P6040_RUN            AT %Q*   :BOOL;    //P6040 Run Command

P7004_RUN            AT %Q*   :BOOL;    //P7004 Run Command
P7010_RUN            AT %Q*   :BOOL;    //P7010 Run Command
P7015_RUN            AT %Q*   :BOOL;    //P7015 Run Command
P7020_RUN            AT %Q*   :BOOL;    //P7020 Run Command
P7025_RUN            AT %Q*   :BOOL;    //P7025 Run Command
P7030_RUN            AT %Q*   :BOOL;    //P7030 Run Command
P7035_RUN            AT %Q*   :BOOL;    //P7035 Run Command
P7045_RUN            AT %Q*   :BOOL;    //P7045 Run Command

 //---------------------------------Motor Feedback-------------------------------------------------

 P6005_Faulted AT %I*: BOOL;		// P6005 Starter Faulted 
 P6015_Faulted AT %I*: BOOL;	    // P6015 Starter Faulted 
 P6020_Faulted AT %I*: BOOL;	    // P6020 Starter Faulted 
 P6025_Faulted AT %I*: BOOL;	    // P6025 Starter Faulted 
 P6030_Faulted AT %I*: BOOL;	    // P6030 Starter Faulted 
 P6035_Faulted AT %I*: BOOL;	    // P6035 Starter Faulted  
 P6040_Faulted AT %I*: BOOL;	    // P6040 Starter Faulted 
 
 P7004_Faulted AT %I*: BOOL;	    // P7004 Starter Faulted 
 P7010_Faulted AT %I*: BOOL;	    // P7010 Starter Faulted 
 P7015_Faulted AT %I*: BOOL;	    // P7015 Starter Faulted 
 P7020_Faulted AT %I*: BOOL;	    // P7020 Starter Faulted 
 P7025_Faulted AT %I*: BOOL;	    // P7025 Starter Faulted 
 P7030_Faulted AT %I*: BOOL;	    // P7035 Starter Faulted 
 P7035_Faulted AT %I*: BOOL;	    // P7035 Starter Faulted 
 P7045_Faulted AT %I*: BOOL;	    // P7045 Starter Faulted  

//---------------------------------Disconnect Status------------------------------------------------- 
{attribute 'OPC.UA.DA' := '1'}
DS_P6005            AT %I*  :BOOL;  //P6005 Disconnect
{attribute 'OPC.UA.DA' := '1'}
DS_P6010            AT %I*  :BOOL;  //P6010 Disconnect
{attribute 'OPC.UA.DA' := '1'}
DS_P6011            AT %I*  :BOOL;  //P6011 Disconnect
{attribute 'OPC.UA.DA' := '1'}
DS_P6015            AT %I*  :BOOL;  //P6015 Disconnect
{attribute 'OPC.UA.DA' := '1'}
DS_P6020            AT %I*  :BOOL;  //P6020 Disconnect
{attribute 'OPC.UA.DA' := '1'}
DS_P6025            AT %I*  :BOOL;  //P6025 Disconnect
{attribute 'OPC.UA.DA' := '1'}
DS_P6030            AT %I*  :BOOL;  //P6030 Disconnect
{attribute 'OPC.UA.DA' := '1'}
DS_P6035            AT %I*  :BOOL;  //P6035 Disconnect
{attribute 'OPC.UA.DA' := '1'}
DS_P6045            AT %I*  :BOOL;  //P6045 Disconnect
{attribute 'OPC.UA.DA' := '1'}
DS_P6040            AT %I*  :BOOL;  //P6040 Disconnect
{attribute 'OPC.UA.DA' := '1'}
DS_P7004            AT %I*  :BOOL;  //P7004 Disconnect
{attribute 'OPC.UA.DA' := '1'}
DS_P7005            AT %I*  :BOOL;  //P7005 Disconnect
{attribute 'OPC.UA.DA' := '1'}
DS_P7010            AT %I*  :BOOL;  //P7010 Disconnect
{attribute 'OPC.UA.DA' := '1'}
DS_P7015            AT %I*  :BOOL;  //P7015 Disconnect
{attribute 'OPC.UA.DA' := '1'}
DS_P7020            AT %I*  :BOOL;  //P7020 Disconnect
{attribute 'OPC.UA.DA' := '1'}
DS_P7025            AT %I*  :BOOL;  //P7025 Disconnect
{attribute 'OPC.UA.DA' := '1'}
DS_P7030            AT %I*  :BOOL;  //P7030 Disconnect
{attribute 'OPC.UA.DA' := '1'}
DS_P7035            AT %I*  :BOOL;  //P7035 Disconnect
{attribute 'OPC.UA.DA' := '1'}
DS_P7040            AT %I*  :BOOL;  //P7040 Disconnect
{attribute 'OPC.UA.DA' := '1'}
DS_P7041            AT %I*  :BOOL;  //P7041 Disconnect
{attribute 'OPC.UA.DA' := '1'}
DS_P7045            AT %I*  :BOOL;  //P7045 Disconnect	
	
//---------------------------------Solenoid Valves------------------------------------------------- 
SV_6181_EXT AT %Q* :BOOL; // GR6040-02 BELT GRIPPER
SV_6211_EXT AT %Q* :BOOL; // GR6040-01 BELT GRIPPER
SV_6301_RET AT %Q* :BOOL; // PI6040-01 PIN STOP
SV_6321_EXT AT %Q* :BOOL; // PI6040-01 PIN STOP
SV_7121_EXT AT %Q* :BOOL; // PU6040-01 PUSH DIVERT
SV_7181_EXT AT %Q* :BOOL; // PU6040-02 PUSH DIVERT
SV_8111_EXT AT %Q* :BOOL; // PU6040-03 PUSH DIVERT
SV_8161_EXT AT %Q* :BOOL; // PU6040-04 "D" GRIPPER

//---------------------------------Encoder------------------------------------------------- 
{attribute 'OPC.UA.DA' := '1'}
	ENC_9021_Raw	AT %I*:	UINT;	// Raw Encoder Value
	{attribute 'OPC.UA.DA' := '1'}
	ENC_9021_OK			: BOOL;
	ENC_9021_Period	AT %I*:	UDINT;	// Encoder Period, channel 1, 100ns resolution
	
	SorterName				: STRING[5];
	
 //---------------------------------WcStates-------------------------------------------------
 	RIO1181_WcState AT %I*				: BOOL;		// Remote IO Block 1181
	RIO4172_WcState AT %I*				: BOOL;		// Remote IO Block 4172
	RIO5151_WcState AT %I*				: BOOL;		// Remote IO Block 5151
	RIO6171_WcState AT %I*				: BOOL;		// Remote IO Block 6171
	RIO7161_WcState AT %I*				: BOOL;		// Remote IO Block 7161
	RIO8181_WcState AT %I*				: BOOL;		// Remote IO Block 8181
	RIO11141_WcState AT %I*				: BOOL;		// Remote IO Block 11141
	RIO12171_WcState AT %I*				: BOOL;		// Remote IO Block 12171
	RIO15181_WcState AT %I*				: BOOL;		// Remote IO Block 15181
	RIO16171_WcState AT %I*				: BOOL;		// Remote IO Block 16171
	BCR_S6040_01_WcState AT %I*			: BOOL;		// Barcode Reader S6040_01
	BCR_S7004_01_WcState AT %I*			: BOOL;		// Barcode Reader S7004_01
	EthernetAdapter_State AT %I*	    : UINT;		// Ethernet Adapter State
 //---------------------------------EAP-------------------------------------------------
//Published
  To205_P6005_IsRunning	AT %Q*:	BOOL; 
  To205_P7045_SendingProduct AT %Q*: BOOL; 
//Subscribed
  From205_P2012_IsRunning AT %I*: BOOL;
  From205_P3130_SendingProduct AT %I*: BOOL;
END_VAR

// ---- GVLs/GVL_Logging.TcGVL
// Comment out attribute to allow direct access to this variable
// {attribute 'qualified_only'} 
VAR_GLOBAL PERSISTENT
	nMessageLogEnable:			UDINT;		// 32 separate log events to enable
	nBarcodeLogEnable:			UDINT;		// 32 separate log events to enable
	nServerLogEnable:			UDINT;		// 32 separate log events to enable, default to enabled, turn off 
	nItemBufferLogEnable:		UDINT;		// 32 separate log events to enable	
	nDivertLogEnable:			UDINT;		// 32 separate log events to enable	
	nSorterLogEnable:			UDINT;		// 32 separate log events to enable	
	nSortBufferLogEnable:		UDINT;		// 32 separate log events to enable	
END_VAR

VAR_GLOBAL CONSTANT
	// To enable a specific log, turn ON the bit associate with that log type in the Enable UDINT 
	// The constants below correspond to the bit number within the UDINT

	// Use E_MessageIds as constants for message logging
	// Barcode Logging
	TRIGGER_PE		:	INT := 0;
	TRIGGER			:	INT := 1;
	BCR_S6040_01_LOG	:	INT := 2;
	BCR_S7004_01_LOG	:	INT := 3;
	
	// Barcode Logging
	BUFFER_LOG	:	INT := 0;	
	// Item Buffer Logging
	ARRIVALS		:	INT := 0;
	TRANSPORT		: 	INT := 1;
	UPDATE			: 	INT := 2;
	// nDivertLogEnable constants
	// Increase for additional Diverts
	DIVERT_DECISION	:	INT := 0;
	DIVERT1			:	INT := 1;
	DIVERT2			:	INT := 2;
	DIVERT3			:	INT := 3;
	DIVERT4			:	INT := 4;
	DIVERT5			:	INT := 5;
	DIVERT6			:	INT := 6;
	DIVERT7			:	INT := 7;
	DIVERT8			:	INT := 8;
	CONFIRM1		:	INT := 16;
	CONFIRM2		:	INT := 17;
	CONFIRM3		:	INT := 18;
	CONFIRM4		:	INT := 19;
	CONFIRM5		:	INT := 20;
	CONFIRM6		:	INT := 21;
	CONFIRM7		:	INT := 22;
	CONFIRM8		:	INT := 23;
	LANEFULL		:	INT := 31;

	// nSorterLogEnable constants
	SORTER_INDUCT		:	INT	:= 0;
	SORTER_INDUCT_PE	:	INT	:= 1;
	SORTER_DIVERTS		:	INT	:= 2;
	SORTER_CONFIRMS		:	INT	:= 3;
	SORTER_DUMP			:	INT	:= 4;
	SORTER_TEMPID		:	INT	:= 5;
	SORTER_HEIGHT_PE	:	INT := 6;
	SORTER_DISCHARGE_PE	:	INT	:= 7;
	SORTER_DESTINATION_LU	:	INT	:= 8;
	// Sorter buffer constants
	BUFFER_ARRIVAL			:	INT := 0;
	BUFFER_MISSINDUCT		: 	INT := 1;
	BUFFER_TEMPINDUCT		:	INT := 2;
	BUFFER_INDUCT			:	INT := 3;
	BUFFER_LATEINDUCT		:	INT := 4;
	BUFFER_REPLACEINDUCT	:	INT := 5;
	BUFFER_UPDATEINDUCT		:	INT := 6;
	BUFFER_UPDATEDEST		:	INT := 7;
	BUFFER_DUMP				:	INT := 8;
	BUFFER_UNASSIGNED		:	INT := 9;
	BUFFER_DESTINDEX		:	INT := 10;
END_VAR

// ---- GVLs/GVL_SorterItems.TcGVL
//{attribute 'qualified_only'}
VAR_GLOBAL
	// Default Destination per Sorter/divert
	P6040_DefaultDestination:		DINT;	// Input default destination update from Host messaging(MsgControl.RECEIVE)

	st_SorterArrivalBufferP6040:		ST_ItemBuffer;		// Output from the Barcode Reader to the sorter
	st_ArrivalFdbkInP6040: 				ST_ItemBufferFdbk;
	st_ArrivalFdbkOutP6040: 			ST_ItemBufferFdbk;

	st_SorterTransportBufferP6040:		ST_ItemBuffer;		// Routing from the ARUP Host to the sorter
	st_TransportFdbkInP6040: 			ST_ItemBufferFdbk;
	st_TransportFdbkOutP6040:	 		ST_ItemBufferFdbk;

	st_SorterUpdateBuffer:				ST_ItemBuffer;  	// Output from the sorter to update the host messaging (MsgControl)
	st_UpdateFdbkIn:					ST_ItemBufferFdbk;
	st_UpdateFdbkOut:					ST_ItemBufferFdbk;

	BlankItem					: ST_Item := (ID := '', UniqueID := 0
													, Destination := 0
													, DestinationIdx := 0
													, Status := E_StatusCode.No_Status
													, ExtStatus := E_StatusCode.No_Status
													, DeviceID := ''
													, MessageType := E_MessageIds.NoMessage_00);

END_VAR

// ---- GVLs/Onsite_Checklist.TcGVL
{attribute 'qualified_only'}
VAR_GLOBAL
	// Air pressure inupt, System Event? , 
	//Set up Air pressure valve
	// Barcode In_EquipID Get from ARUP
	// Link CommFault
	// Setup Full Photoeyes and interlocks 
	// Set up EAP
	
	//Complete?
	// Link CommFault
	// Air pressure event for all solenoids valves 
END_VAR

// ---- POUs/MAIN.TcPOU
PROGRAM MAIN
VAR
	// Data persistence configuration
	rStartPersistentSave 		: R_TRIG; // Rising edge trigger to start persistent data save
	fbWritePersistentData 		: WritePersistentData;
	tonPersistentSave	:	TON := (PT := T#1M);
	tpBroadcastSave		:	TP	:= (PT := T#100MS);
	PLCPersistentSave			AT %Q*	: BOOL;
	ADSPort						:	UINT := 0;
	In_ResetAllMetrics			: 	BOOL;
END_VAR

VAR PERSISTENT
	EAP_205 : ST_EAP_DEVICE ;	
END_VAR

BarCodeReaders();
CommStatus();
Conveyors();
Log_Diverts();
Photoeyes();
ProxSensors();
ServerControl();
Singulation_Control();
Solenoids();
Sorter();
System();
SystemSafety();
P_PulseCountDist();
GVL_IO.INIT := FALSE;


// Reset when Timer is Done
tonPersistentSave(IN := NOT tpBroadcastSave.Q);

// Catch the .Q of the persistent save timer to trigger a save pulse
tpBroadcastSave(IN := tonPersistentSave.Q);
// Set the Persistent save outputs to the .Q of the pulse
PLCPersistentSave := tpBroadcastSave.Q;

// Check for persistent item save
//rStartPersistentSave(CLK := tpBroadcastSave.Q);
// Execute a Persistent save here
// System PORT is 851
fbWritePersistentData(netid:= '', PORT:=851, Start:=tpBroadcastSave.Q, tmout:=T#1S);

// Convert HMI EAP IP Address(es) to correct format
MEMCPY(destAddr    := ADR(EAP_205.Publisher.HMI_IPAddrDisp),srcaddr :=ADR(EAP_205.Publisher.IPAddr), n := 4);
IF ((EAP_205.Publisher.HMI_IPAddrDisp[0] <> EAP_205.Publisher.HMI_IPAddr[0]) AND EAP_205.Publisher.HMI_IPAddr[0] > 0)
   OR ((EAP_205.Publisher.HMI_IPAddrDisp[1] <> EAP_205.Publisher.HMI_IPAddr[1]) AND EAP_205.Publisher.HMI_IPAddr[1] > 0)
   OR ((EAP_205.Publisher.HMI_IPAddrDisp[2] <> EAP_205.Publisher.HMI_IPAddr[2]) AND EAP_205.Publisher.HMI_IPAddr[2] > 0)
   OR ((EAP_205.Publisher.HMI_IPAddrDisp[3] <> EAP_205.Publisher.HMI_IPAddr[3]) AND EAP_205.Publisher.HMI_IPAddr[3] > 0)
   THEN
    MEMCPY(destAddr    := ADR(EAP_205.Publisher.IPAddr),srcaddr :=ADR(EAP_205.Publisher.HMI_IPAddr), n := 4);
END_IF

END_PROGRAM

// ---- POUs/BarCodeReaders.TcPOU
PROGRAM BarCodeReaders
VAR
	BCR_S6040_01: CognexDataMan260;		// P8005 Induct Confirm
	BCR_S7004_01: CognexDataMan260;		// P8010 Location Update
			
		
	Arrival_Item 			: ST_Item;		// Output Item (Bar code read) To Sort PLC
	LastArrival_Item		: ST_Item;		// Last Output Item (Bar code read) To Sort PLC
	ReadID_P6040_Old		: UDINT;

	fb_SorterArrivalBuffer			: FB_ItemBuffer;	// Function to Process the SorterArrivalBuffer
	
	sBcr_S6040_01Log			: STRING;
	tpBcr_S6040_01Trig					: TP;	// Pulse timer for BCR Reader

	rSorterPE					: R_TRIG; 	// Capture the Rising edge of the Sorter BCR PE
	fSorterPE					: F_TRIG; 	// Capture the Falling edge of the Sorter BCR PE
	r_BCR_S6040_01TriggerON			: R_TRIG;
	f_BCR_S6040_01TriggerON			: F_TRIG;

END_VAR

// Create instances of Buffer Processing Functions to initialize the buffers and data
fb_SorterArrivalBuffer.Master := TRUE;

// Setup Logging
fb_SorterArrivalBuffer.LogEntries := .nItemBufferLogEnable.ARRIVALS;

// Setup Buffer Name for Logging
fb_SorterArrivalBuffer.Name := 'SYS ARRIVAL';

fb_SorterArrivalBuffer(st_BufferData := st_SorterArrivalBufferP6040
					, st_BufferFdbkIn := st_ArrivalFdbkInP6040
					, st_BufferFdbkOut => st_ArrivalFdbkOutP6040);

IF GVL_IO.INIT THEN
	fb_SorterArrivalBuffer.Clear();
END_IF
// Reset All Metrics when requested
IF MAIN.In_ResetAllMetrics THEN
	BCR_S6040_01.In_ResetCounts := MAIN.In_ResetAllMetrics;
	BCR_S7004_01.In_ResetCounts := MAIN.In_ResetAllMetrics;
END_IF

// Set up Bar Code Readers
//----------------------------------------P6040--------------------------------------------------------------
BCR_S6040_01.LogEntries := .nBarcodeLogEnable.BCR_S6040_01_LOG;
BCR_S6040_01(
	In_ReadTrig:= PhotoEyes.PE_6261.Out_OnFltrd, 
	In_ResetCounts:= , 
	In_TriggerOnTime := T#20MS ,
	In_EquipID := '00059',
	Out_NewReadTrig=> , 
	Out_ReadString=> , 
	Out_ReadStatus=> ,
	Out_ResultID=>, 
	MisreadCount=> , 
	GoodreadCount=> );
	
BCR_S6040_01.LogEntries := .nBarcodeLogEnable.BCR_S6040_01_LOG;
tpBcr_S6040_01Trig(
	IN := PhotoEyes.PE_6261.Out,
				PT := T#10MS,
				Q =>);
// Capture rising and falling edge Triggers of the Sorter BCR Trigger PE
 rSorterPE(CLK:= PhotoEyes.PE_6261.Out, Q =>);
 fSorterPE(CLK:= PhotoEyes.PE_6261.Out, Q =>);

// Log the rising/falling edge of the Trigger
IF rSorterPE.Q OR fSorterPE.Q THEN
	IF nBarcodeLogEnable.TRIGGER_PE THEN
		// Write to the Error List
		ADSLOGSTR( msgCtrlMask := ADSLOG_MSGTYPE_HINT OR ADSLOG_MSGTYPE_LOG,
			msgFmtStr := 'Sort BCR PE Blocked : %s',
			strArg := BOOL_TO_STRING(PhotoEyes.PE_6261.Out)
			); 
	END_IF
END_IF

// Capture rising and falling edge Triggers of the Sorter BCR Trigger PE
r_BCR_S6040_01TriggerOn(CLK:= BCR_S6040_01.Out_TriggerState, Q =>);
f_BCR_S6040_01TriggerOn(CLK:= BCR_S6040_01.Out_TriggerState, Q =>);

// Log the rising edge of the Trigger
IF r_BCR_S6040_01TriggerOn.Q OR f_BCR_S6040_01TriggerOn.Q THEN
	IF nBarcodeLogEnable.TRIGGER THEN
		// Write to the Error List
		ADSLOGSTR( msgCtrlMask := ADSLOG_MSGTYPE_HINT OR ADSLOG_MSGTYPE_LOG
			, msgFmtStr := 'Sort BCR Trigger : %s'
			, strArg := BOOL_TO_STRING(BCR_S6040_01.Out_TriggerState)); 
	END_IF
END_IF


// Send Read Information to Sorter	
//	Creates Arrival message at sorter
IF ReadID_P6040_Old <> BarCodeReaders.BCR_S6040_01.GoodreadCount THEN
	Arrival_Item.UniqueID := BCR_S6040_01.Out_ResultID;
	Arrival_Item.ID := BCR_S6040_01.Out_ReadString;
	Arrival_Item.Status := E_StatusCode.UpdateRequested;
	Arrival_Item.DeviceID := BArcodeReaders.BCR_S6040_01.In_EquipID;
	Arrival_Item.MessageType := E_MessageIds.Arrival_23;
	Arrival_Item.Destination := MsgControl.DefDestination;
	Arrival_Item.Length := 0;
	LastArrival_Item := Arrival_Item;
	fb_SorterArrivalBuffer.AddItem(Arrival_Item);
	ReadID_P6040_Old := BarCodeReaders.BCR_S6040_01.GoodreadCount;
ELSE 
	Arrival_Item := BlankItem;
	Arrival_Item.Status := E_StatusCode.UpdateRequested;
END_IF	

//----------------------------------------P7004--------------------------------------------------------------	
BCR_S7004_01.LogEntries := .nBarcodeLogEnable.BCR_S7004_01_LOG;
BCR_S7004_01(
	In_ReadTrig:= PhotoEyes.PE_12221.Out_OnFltrd, 
	In_ResetCounts:= , 
	In_TriggerOnTime := T#20MS ,
	In_EquipID := '00062',
	Out_NewReadTrig=> , 
	Out_ReadString=> , 
	Out_ReadStatus=> ,
	Out_ResultID=>, 
	MisreadCount=> , 
	GoodreadCount=> );

END_PROGRAM

// ---- POUs/Photoeyes.TcPOU
{attribute 'OPC.UA.DA' := '1'}

PROGRAM PhotoEyes
VAR
	DebounceOnTime:	TIME := T#500MS;     // Default Value
	DebounceOffTime:	TIME := T#500MS;     // Default Value
	JamDetectTime:	TIME := T#5S;     // Default Value
	TriggerOnTime: TIME :=T#25MS; 
//----------------------------------------Photoeyes-----------------------------------------		
PE_1232:  FB_Photoeye;    //P6005 EXIT PE 
PE_1162:  FB_Photoeye;    //P6010 FULL PE 
PE_1081:  FB_Photoeye;    //P6015 EXIT PE
PE_1231:  FB_Photoeye;    //P6020 FIRE GATE OPEN
PE_1161:  FB_Photoeye;    //P6020 EXIT PE
PE_4121:  FB_Photoeye;    //P6025 EXIT PE
PE_6181:  FB_Photoeye;    //P6040 HEIGHT CHECK HIGH  PE
PE_6201:  FB_Photoeye;    //P6040 HEIGHT CHECK LOW  PE
PE_6261:  FB_Photoeye;    //P6040 SCANNER TRIGGER PE
PE_7171:  FB_Photoeye;    //P6040 SORTER INDUCT
PE_6241:  FB_Photoeye;    //PI6040 PART CLEAR PE
PE_12261:  FB_Photoeye;    //P7004 HEIGHT CHECK PE
PE_12221:  FB_Photoeye;    //P7004 SCANNER TRIGGER PE
PE_16181:  FB_Photoeye;    //P7030 FIRE GATE OPEN PE
PE_4271:  FB_Photoeye;    //PE6030 EXIT PE 
PE_4201:  FB_Photoeye;    //PE6035 EXIT PE 
PE_4071:  FB_Photoeye;    //PE6045 EXIT PE 
PE_6302:  FB_Photoeye;    //PE6040 FULL PE 
PE_12301:  FB_Photoeye;    //PE7005 EXIT PE 
PE_12231:  FB_Photoeye;    //PE7010 EXIT PE 
PE_15121:  FB_Photoeye;    //PE7015 EXIT PE 
PE_15181:  FB_Photoeye;    //PE7020 EXIT PE 
PE_15261:  FB_Photoeye;    //PE7025 EXIT PE 
PE_16111:  FB_Photoeye;    //PE7030 EXIT PE 
PE_16301:  FB_Photoeye;    //PE7035 EXIT PE 
PE_16131:  FB_Photoeye;    //PE7040 EXIT PE 
PE_16201:  FB_Photoeye;    //PE7045 FULL PE 
PE_7151:  FB_Photoeye;    //PU6040-01 JAM PE 
PE_7191:  FB_Photoeye;    //PU6040-01 TRANSFER COMPLETED PE
PE_7211:  FB_Photoeye;    //PU6040-02 JAM PE
PE_7241:  FB_Photoeye;    //PU6040-02 TRANSFER COMPLETED PE
PE_8141:  FB_Photoeye;    //PU6040-03 JAM PE
PE_8171:  FB_Photoeye;    //PU6040-03 TRANSFER COMPLETED PE
PE_8181:  FB_Photoeye;    //PU6040-04 JAM PE 
PE_8221:  FB_Photoeye;    //PU6040-04 TRANSFER COMPLETED PE
PE_8211:  FB_Photoeye;    //PU6040 SORTER DISCHARGE PE
END_VAR

//P6005 EXIT PE   
PE_1232(
   In_Status:= ,
   CFG_PEOKState:= 1,
   CFG_OnDlyTime:= DebounceOnTime,
   CFG_OffDlyTime:= DebounceOffTime,
   CFG_JamDetTime:= JamDetectTime,
   In_Sim:=
);

//P6010 FULL PE   
PE_1162(
   In_Status:= ,
   CFG_PEOKState:= 1,
   CFG_OnDlyTime:= DebounceOnTime,
   CFG_OffDlyTime:= DebounceOffTime,
   CFG_JamDetTime:= JamDetectTime,
   In_Sim:=
);

//P6015 EXIT PE   
PE_1081(
   In_Status:= ,
   CFG_PEOKState:= 1,
   CFG_OnDlyTime:= DebounceOnTime,
   CFG_OffDlyTime:= DebounceOffTime,
   CFG_JamDetTime:= JamDetectTime,
   In_Sim:=
);

//P6020 FIRE GATE OPEN  
PE_1231(
   In_Status:= ,
   CFG_PEOKState:= 1,
   CFG_OnDlyTime:= DebounceOnTime,
   CFG_OffDlyTime:= DebounceOffTime,
   CFG_JamDetTime:= JamDetectTime,
   In_Sim:=
);

//P6020 EXIT PE   
PE_1161(
   In_Status:= ,
   CFG_PEOKState:= 1,
   CFG_OnDlyTime:= DebounceOnTime,
   CFG_OffDlyTime:= DebounceOffTime,
   CFG_JamDetTime:= JamDetectTime,
   In_Sim:=
);

//P6025 EXIT PE   
PE_4121(
   In_Status:= ,
   CFG_PEOKState:= 1,
   CFG_OnDlyTime:= DebounceOnTime,
   CFG_OffDlyTime:= DebounceOffTime,
   CFG_JamDetTime:= JamDetectTime,
   In_Sim:=
);

//P6040 HEIGHT CHECK HIGH  PE
PE_6181(
   In_Status:= ,
   CFG_PEOKState:= 1,
   CFG_OnDlyTime:= DebounceOnTime,
   CFG_OffDlyTime:= DebounceOffTime,
   CFG_JamDetTime:= JamDetectTime,
   In_Sim:=
);

//P6040 HEIGHT CHECK LOW  PE
PE_6201(
   In_Status:= ,
   CFG_PEOKState:= 1,
   CFG_OnDlyTime:= DebounceOnTime,
   CFG_OffDlyTime:= DebounceOffTime,
   CFG_JamDetTime:= JamDetectTime,
   In_Sim:=
);

//P6040 SCANNER TRIGGER PE  
PE_6261(
   In_Status:= ,
   CFG_PEOKState:= 1,
   CFG_OnDlyTime:= TriggerOnTime,
   CFG_OffDlyTime:= DebounceOffTime,
   CFG_JamDetTime:= JamDetectTime,
   In_Sim:=
);

//P6040 SORTER INDUCT 
PE_7171(
   In_Status:= ,
   CFG_PEOKState:= 1,
   CFG_OnDlyTime:= DebounceOnTime,
   CFG_OffDlyTime:= DebounceOffTime,
   CFG_JamDetTime:= JamDetectTime,
   In_Sim:=
);

//PI6040 PART CLEAR PE  
PE_6241(
   In_Status:= ,
   CFG_PEOKState:= 1,
   CFG_OnDlyTime:= DebounceOnTime,
   CFG_OffDlyTime:= DebounceOffTime,
   CFG_JamDetTime:= JamDetectTime,
   In_Sim:=
);

//P7004 HEIGHT CHECK   
PE_12261(
   In_Status:= ,
   CFG_PEOKState:= 1,
   CFG_OnDlyTime:= DebounceOnTime,
   CFG_OffDlyTime:= DebounceOffTime,
   CFG_JamDetTime:= JamDetectTime,
   In_Sim:=
);

//P7004 SCANNER TRIGGER   
PE_12221(
   In_Status:= ,
   CFG_PEOKState:= 1,
   CFG_OnDlyTime:= TriggerOnTime,
   CFG_OffDlyTime:= DebounceOffTime,
   CFG_JamDetTime:= JamDetectTime,
   In_Sim:=
);

//P7030 FIRE GATE OPEN  
PE_16181(
   In_Status:= ,
   CFG_PEOKState:= 1,
   CFG_OnDlyTime:= DebounceOnTime,
   CFG_OffDlyTime:= DebounceOffTime,
   CFG_JamDetTime:= JamDetectTime,
   In_Sim:=
);

//PE6030 EXIT PE   
PE_4271(
   In_Status:= ,
   CFG_PEOKState:= 1,
   CFG_OnDlyTime:= DebounceOnTime,
   CFG_OffDlyTime:= DebounceOffTime,
   CFG_JamDetTime:= JamDetectTime,
   In_Sim:=
);

//PE6035 EXIT PE   
PE_4201(
   In_Status:= ,
   CFG_PEOKState:= 1,
   CFG_OnDlyTime:= DebounceOnTime,
   CFG_OffDlyTime:= DebounceOffTime,
   CFG_JamDetTime:= JamDetectTime,
   In_Sim:=
);

//PE6045 FULL PE   
PE_4071(
   In_Status:= ,
   CFG_PEOKState:= 1,
   CFG_OnDlyTime:= DebounceOnTime,
   CFG_OffDlyTime:= DebounceOffTime,
   CFG_JamDetTime:= JamDetectTime,
   In_Sim:=
);

//PE6045 FULL PE   
PE_6302(
   In_Status:= ,
   CFG_PEOKState:= 1,
   CFG_OnDlyTime:= DebounceOnTime,
   CFG_OffDlyTime:= DebounceOffTime,
   CFG_JamDetTime:= JamDetectTime,
   In_Sim:=
);

//PE7005 EXIT PE   
PE_12301(
   In_Status:= ,
   CFG_PEOKState:= 1,
   CFG_OnDlyTime:= DebounceOnTime,
   CFG_OffDlyTime:= DebounceOffTime,
   CFG_JamDetTime:= JamDetectTime,
   In_Sim:=
);

//PE7010 EXIT PE   
PE_12231(
   In_Status:= ,
   CFG_PEOKState:= 1,
   CFG_OnDlyTime:= DebounceOnTime,
   CFG_OffDlyTime:= DebounceOffTime,
   CFG_JamDetTime:= JamDetectTime,
   In_Sim:=
);

//PE7015 EXIT PE   
PE_15121(
   In_Status:= ,
   CFG_PEOKState:= 1,
   CFG_OnDlyTime:= DebounceOnTime,
   CFG_OffDlyTime:= DebounceOffTime,
   CFG_JamDetTime:= JamDetectTime,
   In_Sim:=
);

//PE7020 EXIT PE   
PE_15181(
   In_Status:= ,
   CFG_PEOKState:= 1,
   CFG_OnDlyTime:= DebounceOnTime,
   CFG_OffDlyTime:= DebounceOffTime,
   CFG_JamDetTime:= JamDetectTime,
   In_Sim:=
);

//PE7025 EXIT PE   
PE_15261(
   In_Status:= ,
   CFG_PEOKState:= 1,
   CFG_OnDlyTime:= DebounceOnTime,
   CFG_OffDlyTime:= DebounceOffTime,
   CFG_JamDetTime:= JamDetectTime,
   In_Sim:=
);

//PE7030 EXIT PE   
PE_16111(
   In_Status:= ,
   CFG_PEOKState:= 1,
   CFG_OnDlyTime:= DebounceOnTime,
   CFG_OffDlyTime:= DebounceOffTime,
   CFG_JamDetTime:= JamDetectTime,
   In_Sim:=
);

//PE7035 EXIT PE   
PE_16301(
   In_Status:= ,
   CFG_PEOKState:= 1,
   CFG_OnDlyTime:= DebounceOnTime,
   CFG_OffDlyTime:= DebounceOffTime,
   CFG_JamDetTime:= JamDetectTime,
   In_Sim:=
);

//PE7040 EXIT PE   
PE_16131(
   In_Status:= ,
   CFG_PEOKState:= 1,
   CFG_OnDlyTime:= DebounceOnTime,
   CFG_OffDlyTime:= DebounceOffTime,
   CFG_JamDetTime:= JamDetectTime,
   In_Sim:=
);

//PE7045 EXIT PE   
PE_16201(
   In_Status:= ,
   CFG_PEOKState:= 1,
   CFG_OnDlyTime:= DebounceOnTime,
   CFG_OffDlyTime:= DebounceOffTime,
   CFG_JamDetTime:= JamDetectTime,
   In_Sim:=
);

//PU6040-01 JAM PE   
PE_7151(
   In_Status:= Conveyors.P6040_Status.Sts_IsRunning ,
   CFG_PEOKState:= 1,
   CFG_OnDlyTime:= DebounceOnTime,
   CFG_OffDlyTime:= DebounceOffTime,
   CFG_JamDetTime:= JamDetectTime,
   In_Sim:=
);

//PU6040-01 TRANSFER COMPLETED   
PE_7191(
   In_Status:= ,
   CFG_PEOKState:= 1,
   CFG_OnDlyTime:= DebounceOnTime,
   CFG_OffDlyTime:= DebounceOffTime,
   CFG_JamDetTime:= JamDetectTime,
   In_Sim:=
);

//PU6040-02 JAM PE   
PE_7211(
   In_Status:= Conveyors.P6040_Status.Sts_IsRunning ,
   CFG_PEOKState:= 1,
   CFG_OnDlyTime:= DebounceOnTime,
   CFG_OffDlyTime:= DebounceOffTime,
   CFG_JamDetTime:= JamDetectTime,
   In_Sim:=
);

//PU6040-02 TRANSFER COMPLETED   
PE_7241(
   In_Status:= ,
   CFG_PEOKState:= 1,
   CFG_OnDlyTime:= DebounceOnTime,
   CFG_OffDlyTime:= DebounceOffTime,
   CFG_JamDetTime:= JamDetectTime,
   In_Sim:=
);

//PU6040-03 JAM PE   
PE_8141(
   In_Status:= Conveyors.P6040_Status.Sts_IsRunning,
   CFG_PEOKState:= 1,
   CFG_OnDlyTime:= DebounceOnTime,
   CFG_OffDlyTime:= DebounceOffTime,
   CFG_JamDetTime:= JamDetectTime,
   In_Sim:=
);

//PU6040-03 TRANSFER COMPLETED   
PE_8171(
   In_Status:= ,
   CFG_PEOKState:= 1,
   CFG_OnDlyTime:= DebounceOnTime,
   CFG_OffDlyTime:= DebounceOffTime,
   CFG_JamDetTime:= JamDetectTime,
   In_Sim:=
);

//PU6040-04 JAM PE   
PE_8181(
   In_Status:= Conveyors.P6040_Status.Sts_IsRunning ,
   CFG_PEOKState:= 1,
   CFG_OnDlyTime:= DebounceOnTime,
   CFG_OffDlyTime:= DebounceOffTime,
   CFG_JamDetTime:= JamDetectTime,
   In_Sim:=
);

//PU6040-04 TRANSFER COMPLETED   
PE_8221(
   In_Status:= ,
   CFG_PEOKState:= 1,
   CFG_OnDlyTime:= DebounceOnTime,
   CFG_OffDlyTime:= DebounceOffTime,
   CFG_JamDetTime:= JamDetectTime,
   In_Sim:=
);

//PU6040 SORTER DISCHARGE  
PE_8211(
   In_Status:= ,
   CFG_PEOKState:= 1,
   CFG_OnDlyTime:= DebounceOnTime,
   CFG_OffDlyTime:= DebounceOffTime,
   CFG_JamDetTime:= JamDetectTime,
   In_Sim:=
);

END_PROGRAM

// ---- POUs/Conveyors.TcPOU
PROGRAM Conveyors
VAR
	DefaultVelocity: INT := 1675;
	DefaultVelocityThreshold: INT := 500;
	ResetAllDrives: BOOL;
	
//Conveyors Incoming 6000 (Blue line)
//Transport
//----------------------------------------P6005--------------------------------------------------------------
   cfgP6005Label:	STRING(20) :=  'P6005';
   cfgP6005SleepTime:	TIME := T#180S;
   cfgP6005JamDetectTime:	TIME := T#30S;
   P6005SleepWakeTrig: ARRAY[1..5] OF BOOL;
   P6005: FB_CnvyrCnfig_1;
   P6005_StatePB: ST_StateCntrlPB;
   P6005_Status : ST_EquipmentStatus;
//Spiral
//----------------------------------------P6010--------------------------------------------------------------
   cfgP6010Label:	STRING(20) :=  'P6010';
   cfgP6010SleepTime:	TIME := T#180S;
   cfgP6010JamDetectTime:	TIME := T#30S;
   P6010SleepWakeTrig: ARRAY[1..5] OF BOOL;
   P6010: FB_CnvyrCnfig_1;
   P6010_StatePB: ST_StateCntrlPB;
   P6010_Status : ST_EquipmentStatus;
   P6010_VFD	:	VFD;
   Test_VFD_P6010: BOOL;

//Transport
//----------------------------------------P6015--------------------------------------------------------------
   cfgP6015Label:	STRING(20) :=  'P6015';
   cfgP6015SleepTime:	TIME := T#180S;
   cfgP6015JamDetectTime:	TIME := T#30S;
   P6015SleepWakeTrig: ARRAY[1..5] OF BOOL;
   P6015: FB_CnvyrCnfig_1;
   P6015_StatePB: ST_StateCntrlPB;
   P6015_Status : ST_EquipmentStatus;
//----------------------------------------P6020--------------------------------------------------------------
   cfgP6020Label:	STRING(20) :=  'P6020';
   cfgP6020SleepTime:	TIME := T#180S;
   cfgP6020JamDetectTime:	TIME := T#30S;
   P6020SleepWakeTrig: ARRAY[1..5] OF BOOL;
   P6020: FB_CnvyrCnfig_1;
   P6020_StatePB: ST_StateCntrlPB;
   P6020_Status : ST_EquipmentStatus;
//----------------------------------------P6025--------------------------------------------------------------
   cfgP6025Label:	STRING(20) :=  'P6025';
   cfgP6025SleepTime:	TIME := T#180S;
   cfgP6025JamDetectTime:	TIME := T#30S;
   P6025SleepWakeTrig: ARRAY[1..5] OF BOOL;
   P6025: FB_CnvyrCnfig_1;
   P6025_StatePB: ST_StateCntrlPB;
   P6025_Status : ST_EquipmentStatus;
//----------------------------------------P6030--------------------------------------------------------------
   cfgP6030Label:	STRING(20) :=  'P6030';
   cfgP6030SleepTime:	TIME := T#180S;
   cfgP6030JamDetectTime:	TIME := T#30S;
   P6030SleepWakeTrig: ARRAY[1..5] OF BOOL;
   P6030: FB_CnvyrCnfig_1;
   P6030_StatePB: ST_StateCntrlPB;
   P6030_Status : ST_EquipmentStatus;
//----------------------------------------P6035--------------------------------------------------------------
   cfgP6035Label:	STRING(20) :=  'P6035';
   cfgP6035SleepTime:	TIME := T#180S;
   cfgP6035JamDetectTime:	TIME := T#30S;
   P6035SleepWakeTrig: ARRAY[1..5] OF BOOL;
   P6035: FB_CnvyrCnfig_1;
   P6035_StatePB: ST_StateCntrlPB;
   P6035_Status : ST_EquipmentStatus;
//Spiral
//----------------------------------------P6045--------------------------------------------------------------
   cfgP6045Label:	STRING(20) :=  'P6045';
   cfgP6045SleepTime:	TIME := T#180S;
   cfgP6045JamDetectTime:	TIME := T#30S;
   P6045SleepWakeTrig: ARRAY[1..5] OF BOOL;
   P6045: FB_CnvyrCnfig_1;
   P6045_StatePB: ST_StateCntrlPB;
   P6045_Status : ST_EquipmentStatus;
   P6045_VFD	:	VFD;
   Test_VFD_P6045: BOOL;
//Sorter
//----------------------------------------P6040--------------------------------------------------------------
   cfgP6040Label:	STRING(20) :=  'P6040';
   cfgP6040SleepTime:	TIME := T#180S;
   cfgP6040JamDetectTime:	TIME := T#5S;
   P6040SleepWakeTrig: ARRAY[1..5] OF BOOL;
   P6040: FB_CnvyrCnfig_1;
   P6040_StatePB: ST_StateCntrlPB;
   P6040_Status : ST_EquipmentStatus;

//Conveyors Outgoing 7000 (Orange line)
//Loading Zone
//----------------------------------------P7004--------------------------------------------------------------
   cfgP7004Label:	STRING(20) :=  'P7004';
   cfgP7004SleepTime:	TIME := T#180S;
   cfgP7004JamDetectTime:	TIME := T#30S;
   P7004SleepWakeTrig: ARRAY[1..5] OF BOOL;
   P7004: FB_CnvyrCnfig_1;
   P7004_StatePB: ST_StateCntrlPB;
   P7004_Status : ST_EquipmentStatus;
//Spiral
//----------------------------------------P7005--------------------------------------------------------------
   cfgP7005Label:	STRING(20) :=  'P7005';
   cfgP7005SleepTime:	TIME := T#180S;
   cfgP7005JamDetectTime:	TIME := T#30S;
   P7005SleepWakeTrig: ARRAY[1..5] OF BOOL;
   P7005: FB_CnvyrCnfig_1;
   P7005_StatePB: ST_StateCntrlPB;
   P7005_Status : ST_EquipmentStatus;
   P7005_VFD	:	VFD;
   Test_VFD_P7005: BOOL;
   P7005_ResetWakeTmr : TON ; //Timer for holding the reset button to wake up Infeed Conveyor
//Transport
//----------------------------------------P7010--------------------------------------------------------------
   cfgP7010Label:	STRING(20) :=  'P7010';
   cfgP7010SleepTime:	TIME := T#180S;
   cfgP7010JamDetectTime:	TIME := T#30S;
   P7010SleepWakeTrig: ARRAY[1..5] OF BOOL;
   P7010: FB_CnvyrCnfig_1;
   P7010_StatePB: ST_StateCntrlPB;
   P7010_Status : ST_EquipmentStatus;
//----------------------------------------P7015--------------------------------------------------------------
   cfgP7015Label:	STRING(20) :=  'P7015';
   cfgP7015SleepTime:	TIME := T#180S;
   cfgP7015JamDetectTime:	TIME := T#30S;
   P7015SleepWakeTrig: ARRAY[1..5] OF BOOL;
   P7015: FB_CnvyrCnfig_1;
   P7015_StatePB: ST_StateCntrlPB;
   P7015_Status : ST_EquipmentStatus;
//----------------------------------------P7020--------------------------------------------------------------
   cfgP7020Label:	STRING(20) :=  'P7020';
   cfgP7020SleepTime:	TIME := T#180S;
   cfgP7020JamDetectTime:	TIME := T#30S;
   P7020SleepWakeTrig: ARRAY[1..5] OF BOOL;
   P7020: FB_CnvyrCnfig_1;
   P7020_StatePB: ST_StateCntrlPB;
   P7020_Status : ST_EquipmentStatus;
//----------------------------------------P7025--------------------------------------------------------------
   cfgP7025Label:	STRING(20) :=  'P7025';
   cfgP7025SleepTime:	TIME := T#180S;
   cfgP7025JamDetectTime:	TIME := T#30S;
   P7025SleepWakeTrig: ARRAY[1..5] OF BOOL;
   P7025: FB_CnvyrCnfig_1;
   P7025_StatePB: ST_StateCntrlPB;
   P7025_Status : ST_EquipmentStatus;
//----------------------------------------P7030--------------------------------------------------------------
   cfgP7030Label:	STRING(20) :=  'P7030';
   cfgP7030SleepTime:	TIME := T#180S;
   cfgP7030JamDetectTime:	TIME := T#30S;
   P7030SleepWakeTrig: ARRAY[1..5] OF BOOL;
   P7030: FB_CnvyrCnfig_1;
   P7030_StatePB: ST_StateCntrlPB;
   P7030_Status : ST_EquipmentStatus;
//----------------------------------------P7035--------------------------------------------------------------
   cfgP7035Label:	STRING(20) :=  'P7035';
   cfgP7035SleepTime:	TIME := T#180S;
   cfgP7035JamDetectTime:	TIME := T#30S;
   P7035SleepWakeTrig: ARRAY[1..5] OF BOOL;
   P7035: FB_CnvyrCnfig_1;
   P7035_StatePB: ST_StateCntrlPB;
   P7035_Status : ST_EquipmentStatus;
//Spiral
//----------------------------------------P7040--------------------------------------------------------------
   cfgP7040Label:	STRING(20) :=  'P7040';
   cfgP7040SleepTime:	TIME := T#180S;
   cfgP7040JamDetectTime:	TIME := T#30S;
   P7040SleepWakeTrig: ARRAY[1..5] OF BOOL;
   P7040: FB_CnvyrCnfig_1;
   P7040_StatePB: ST_StateCntrlPB;
   P7040_Status : ST_EquipmentStatus;
   P7040_VFD	:	VFD;
   Test_VFD_P7040: BOOL;

//Transport
//----------------------------------------P7045--------------------------------------------------------------
   cfgP7045Label:	STRING(20) :=  'P7045';
   cfgP7045SleepTime:	TIME := T#180S;
   cfgP7045JamDetectTime:	TIME := T#30S;
   P7045SleepWakeTrig: ARRAY[1..5] OF BOOL;
   P7045: FB_CnvyrCnfig_1;
   P7045_StatePB: ST_StateCntrlPB;
   P7045_Status : ST_EquipmentStatus;
END_VAR

VAR PERSISTENT
//Conveyors Incoming 6000 (Blue line)
//Transport
//----------------------------------------P6005--------------------------------------------------------------
{attribute 'OPC.UA.DA' := '1'}
cfgP6005IntlksArry: ARRAY [0..15] OF ST_CfgEvents := [
   (Description := 'Exit PE/Downstream MTR status' , DeviceLabel := '' , OKState := TRUE),   //DeviceLabel: Exit PE downstream
   (Description := 'System Interlocks' , DeviceLabel := '', OKState := TRUE, StopCode := E_StopCodes.SystemStop),
   13(())];
{attribute 'OPC.UA.DA' := '1'}
cfgP6005EvntsArry: ARRAY [0..15] OF ST_CfgEvents := [
   (Description := 'Jam Detected', DeviceLabel := '', LatchRequired := TRUE, OKState := FALSE, StopCode := E_StopCodes.ProductJam),   //DeviceLabel: Jam PE
   (),
   (Description := 'Disconnect', DeviceLabel := 'DS6005', OKState := TRUE, StopCode := E_StopCodes.DisconnectState),   //DeviceLabel: Motor Disconnect
   (Description := 'System Fault', DeviceLabel := 'System', OKState := TRUE, FaultWarn:= TRUE, StopCode := E_StopCodes.SystemStop),
   (Description := 'Fire Door Closed', DeviceLabel := 'PE_16181', OKState := TRUE, FaultWarn:= TRUE, StopCode := E_StopCodes.SystemStop),
   (Description := 'RIO1181 Comm Fault', DeviceLabel := 'RIO1181', OKState := TRUE, FaultWarn:= TRUE, StopCode := E_StopCodes.FieldIOFLT),
   (Description := 'Motor Faulted', DeviceLabel := 'P6005', OKState := FALSE, StopCode := E_StopCodes.MotorOL),
   9(())];
//Spiral
//----------------------------------------P6010--------------------------------------------------------------
{attribute 'OPC.UA.DA' := '1'}
cfgP6010IntlksArry: ARRAY [0..15] OF ST_CfgEvents := [
   (Description := 'Exit PE/Downstream MTR status' , DeviceLabel := '' , OKState := TRUE),   //DeviceLabel: Exit PE downstream
   (Description := 'System Interlocks' , DeviceLabel := '', OKState := TRUE, StopCode := E_StopCodes.SystemStop),
   13(())];
{attribute 'OPC.UA.DA' := '1'}
cfgP6010EvntsArry: ARRAY [0..15] OF ST_CfgEvents := [
   (Description := 'Jam Detected', DeviceLabel := '', LatchRequired := TRUE, OKState := FALSE, StopCode := E_StopCodes.ProductJam),   //DeviceLabel: Jam PE
   (),
   (Description := 'Disconnect', DeviceLabel := 'DS6010', OKState := TRUE, StopCode := E_StopCodes.DisconnectState),   //DeviceLabel: Motor Disconnect
   (Description := 'System Fault', DeviceLabel := 'System', OKState := TRUE, FaultWarn:= TRUE, StopCode := E_StopCodes.SystemStop),
   (Description := 'RIO1181 Comm Fault', DeviceLabel := 'RIO1181', OKState := TRUE, FaultWarn:= TRUE, StopCode := E_StopCodes.FieldIOFLT),
   (Description := 'VFD State Not OK', DeviceLabel := 'P6010', OKState := TRUE, StopCode := E_StopCodes.VFD_Fault),
   10(())];

